// TIA Portal project "2020冬完善底层" (V15)

(* hardware
DEVICE "S7-1200 station_1"  S7-1200 Station
   slot 0: "Rack_0"  S7-1200 Rack  Rack  V1.0
   slot 1: "PLC_1"  CPU 1212C DC/DC/DC  6ES7 212-1AE40-0XB0  V4.2
   slot 3: "AQ 1x12BIT_1"  AQ1 signal board  6ES7 232-4HA30-0XB0  V1.0
DEVICE "S7-1200 station_2"  S7-1200 Station
   slot 0: "Rack_0"  S7-1200 Rack  Rack  V1.0
   slot 1: "PLC_2"  CPU 1212C DC/DC/DC  6ES7 212-1AE40-0XB0  V4.2
   slot 3: "AQ 1x12BIT_1"  AQ1 signal board  6ES7 232-4HA30-0XB0  V1.0
DEVICE "S7-1200 station_3"  S7-1200 Station
   slot 0: "Rack_0"  S7-1200 Rack  Rack  V1.0
   slot 1: "PLC_3"  CPU 1212C DC/DC/DC  6ES7 212-1AE40-0XB0  V4.2
   slot 3: "AQ 1x12BIT_1"  AQ1 signal board  6ES7 232-4HA30-0XB0  V1.0
DEVICE "S7-1200 station_4"  S7-1200 Station
   slot 0: "Rack_0"  S7-1200 Rack  Rack  V1.0
   slot 1: "PLC_4"  CPU 1212C DC/DC/DC  6ES7 212-1AE40-0XB0  V4.2
   slot 3: "AQ 1x12BIT_1"  AQ1 signal board  6ES7 232-4HA30-0XB0  V1.0
*)

// ===== PLC "PLC_1"  CPU 1212C DC/DC/DC =====

VAR_GLOBAL   // PLC tag table "默认变量表"
   "JogForward" AT %I200.0 : Bool;
   "JogBackward" AT %I200.1 : Bool;
   "driver" AT %I200.2 : Bool;
   "Anlonage input" AT %IW208 : Word;
   "R驱动编码器值" AT %ID1000 : DWord;
   "position" AT %IW202 : Word;
   "velecity" AT %ID204 : DWord;
   "R旋转编码器值" AT %ID1008 : DWord;
   "spin" AT %I200.3 : Bool;
   "轴_1_脉冲" AT %Q0.0 : Bool;
   "轴_1_方向" AT %Q0.1 : Bool;
   "AQ电压模拟量输出口" AT %QW80 : Word;
   "旋转编码器值保持" AT %MD0 : DWord;
   "一次写入" AT %M5.0 : Bool;
   "旋转速度转换real" AT %MD24 : Real;
   "原地转向临时速度" AT %MD100 : DWord;
   "原地转向-二号车轮转换" AT %MD104 : Real;
   "原地转向-四号车轮转换" AT %MD108 : Real;
   "原地转向-三号车轮转换" AT %MD112 : Real;
   "二号车轮方向判断继电器" AT %M118.0 : Bool;
   "三号车轮方向判断继电器" AT %M118.1 : Bool;
   "四号车轮方向判断继电器" AT %M118.2 : Bool;
END_VAR

DATA_BLOCK "数据块_1"   // DB1
{ S7_Optimized_Access := 'FALSE' }
VERSION : 0.1
   VAR
      一号车轮旋转开关 : Bool;
      一号车轮直行开关 : Bool;
      一号车轮目标旋转位置 : Word;
      一号车论旋转速度 : DWord;
      "一号车轮直行模拟量（已校准）" : Word;
      二号车轮旋转开关 : Bool;
      二号车轮直行开关 : Bool;
      二号车轮目标旋转位置 : Word;
      二号车轮旋转速度 : DWord;
      "二号车轮直行模拟量（已校准）" : Word;
      三号车轮旋转开关 : Bool;
      三号车轮直行开关 : Bool;
      三号车轮目标旋转位置 : Word;
      三号车轮旋转速度 : DWord;
      "三号车轮直行模拟量（已校准）" : Word;
      四号车轮旋转开关 : Bool;
      四号车轮直行开关 : Bool;
      四号车轮目标旋转位置 : Word;
      四号车轮旋转速度 : DWord;
      "四号车轮直行模拟量（已校准）" : Word;
      "转弯半径（未用）" : Int;
      运动模式 : Byte;
      一号车轮转角编码器读取 : DWord;
      一号车轮速度编码器读取 : DWord;
      二号车轮转角编码器读取 : DWord;
      二号车轮速度编码器读取 : DWord;
      三号车轮转角编码器读取 : DWord;
      三号车轮速度编码器读取 : DWord;
      四号车轮转角编码器读取 : DWord;
      四号车轮速度编码器读取 : DWord;
      一号车轮写入速度 : Word;
      二号车轮写入速度 : Word;
      三号车轮写入速度 : Word;
      四号车轮写入速度 : Word;
   END_VAR
BEGIN
END_DATA_BLOCK

DATA_BLOCK "轴_1"   // DB2, Motion_DB
{ S7_Optimized_Access := 'TRUE' }
AUTHOR : SIMATIC
FAMILY : BasicMC
NAME : TO_PosAx
VERSION : 6.0
// stored: InstanceOfName TO_PositioningAxis
"TO_PositioningAxis"
BEGIN
   // Axis.OnlinePtoModeCU = 16#0000_0002
   // Axis.DirectionOutputEnabledCU = TRUE
   // Axis.SelectedChannel2EnumCU = %Q0.1
   // Axis.SelectedChannel1EnumCU = %Q0.0
   // Pulse.MinDeltaDeltaFrequencyCU = 0.004
   // Pulse.MaxDeltaDeltaFrequencyCU = 1.0E+10
   // Pulse.MinDeltaFrequencyCU = 0.005
   // Pulse.MaxDeltaFrequencyCU = 9.5E+9
   // Pulse.MinFrequencyCU = 1.0
   // Pulse.MaxFrequencyCU = 100000.0
   // Pulse.OutputSourceCU = 16#0000_0000
   // Axis.SelectPTO = 0
END_DATA_BLOCK

FUNCTION "WRITE设备数据传递到各个设备" : Void   // FC1, SCL
{ S7_Optimized_Access := 'TRUE' }
VERSION : 0.1
BEGIN
   POKE_BLK(area_src := 16#84,
            dbNumber_src := 1,
            byteOffset_src := 10,
            area_dest := 16#82,
            dbNumber_dest := 0,
            byteOffset_dest := 200,
            count := 30);
   POKE_BLK(area_src := 16#84,
            dbNumber_src := 1,
            byteOffset_src := 2,
            area_dest := 16#81,
            dbNumber_dest := 0,
            byteOffset_dest := 202,
            count := 8);
   POKE_BLK(area_src:=16#81,
            dbNumber_src:=0,
            byteOffset_src:=300,
            area_dest:=16#84,
            dbNumber_dest:=1,
            byteOffset_dest:=52,
            count:=24);
END_FUNCTION

FUNCTION "模式选择" : Void   // FC2, LAD
{ S7_Optimized_Access := 'TRUE' }
VERSION : 0.1
BEGIN

REGION Network 1
   // 运动模式，01为四轮02为四轮异向03为前轮04为原地
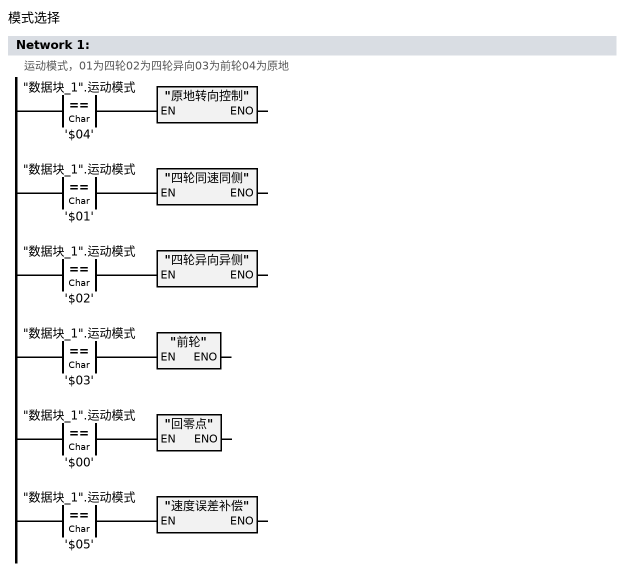
   RUNG wire#powerrail
      { S7_Templates := "SrcType := Char" } EQ_Contact(in1 := "数据块_1".运动模式, in2 := '$04')
      "原地转向控制"()
   END_RUNG
   RUNG wire#powerrail
      { S7_Templates := "SrcType := Char" } EQ_Contact(in1 := "数据块_1".运动模式, in2 := '$01')
      "四轮同速同侧"()
   END_RUNG
   RUNG wire#powerrail
      { S7_Templates := "SrcType := Char" } EQ_Contact(in1 := "数据块_1".运动模式, in2 := '$02')
      "四轮异向异侧"()
   END_RUNG
   RUNG wire#powerrail
      { S7_Templates := "SrcType := Char" } EQ_Contact(in1 := "数据块_1".运动模式, in2 := '$03')
      "前轮"()
   END_RUNG
   RUNG wire#powerrail
      { S7_Templates := "SrcType := Char" } EQ_Contact(in1 := "数据块_1".运动模式, in2 := '$00')
      "回零点"()
   END_RUNG
   RUNG wire#powerrail
      { S7_Templates := "SrcType := Char" } EQ_Contact(in1 := "数据块_1".运动模式, in2 := '$05')
      "速度误差补偿"()
   END_RUNG
   // the same network as SCL:
   IF "数据块_1".运动模式 = '$04' THEN "原地转向控制"(); END_IF;
   IF "数据块_1".运动模式 = '$01' THEN "四轮同速同侧"(); END_IF;
   IF "数据块_1".运动模式 = '$02' THEN "四轮异向异侧"(); END_IF;
   IF "数据块_1".运动模式 = '$03' THEN "前轮"(); END_IF;
   IF "数据块_1".运动模式 = '$00' THEN "回零点"(); END_IF;
   IF "数据块_1".运动模式 = '$05' THEN "速度误差补偿"(); END_IF;
END_REGION
END_FUNCTION

FUNCTION "原地转向控制" : Void   // FC3, LAD
{ S7_Optimized_Access := 'TRUE' }
VERSION : 0.1
BEGIN

REGION Network 1
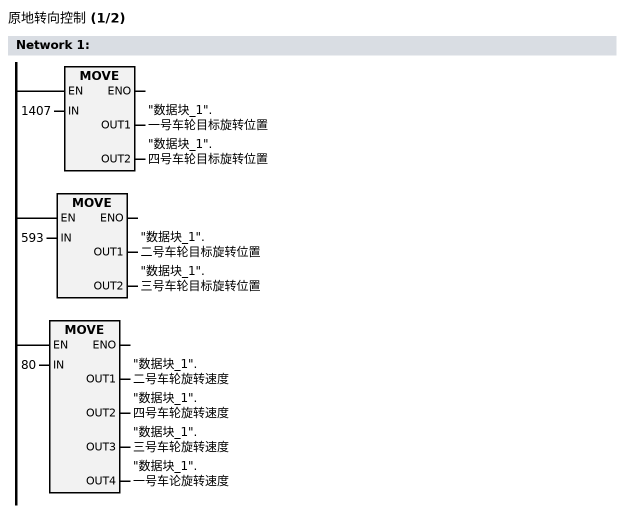
   RUNG wire#powerrail
      Move(in := 1407, out1 => "数据块_1".一号车轮目标旋转位置, out2 => "数据块_1".四号车轮目标旋转位置)
   END_RUNG
   RUNG wire#powerrail
      Move(in := 593, out1 => "数据块_1".二号车轮目标旋转位置, out2 => "数据块_1".三号车轮目标旋转位置)
   END_RUNG
   RUNG wire#powerrail
      Move(in := 80, out1 => "数据块_1".二号车轮旋转速度, out2 => "数据块_1".四号车轮旋转速度, out3 => "数据块_1".三号车轮旋转速度, out4 => "数据块_1".一号车论旋转速度)
   END_RUNG
   // the same network as SCL:
   "数据块_1".一号车轮目标旋转位置 := 1407;
   "数据块_1".四号车轮目标旋转位置 := 1407;
   "数据块_1".二号车轮目标旋转位置 := 593;
   "数据块_1".三号车轮目标旋转位置 := 593;
   "数据块_1".二号车轮旋转速度 := 80;
   "数据块_1".四号车轮旋转速度 := 80;
   "数据块_1".三号车轮旋转速度 := 80;
   "数据块_1".一号车论旋转速度 := 80;
END_REGION

REGION Network 2
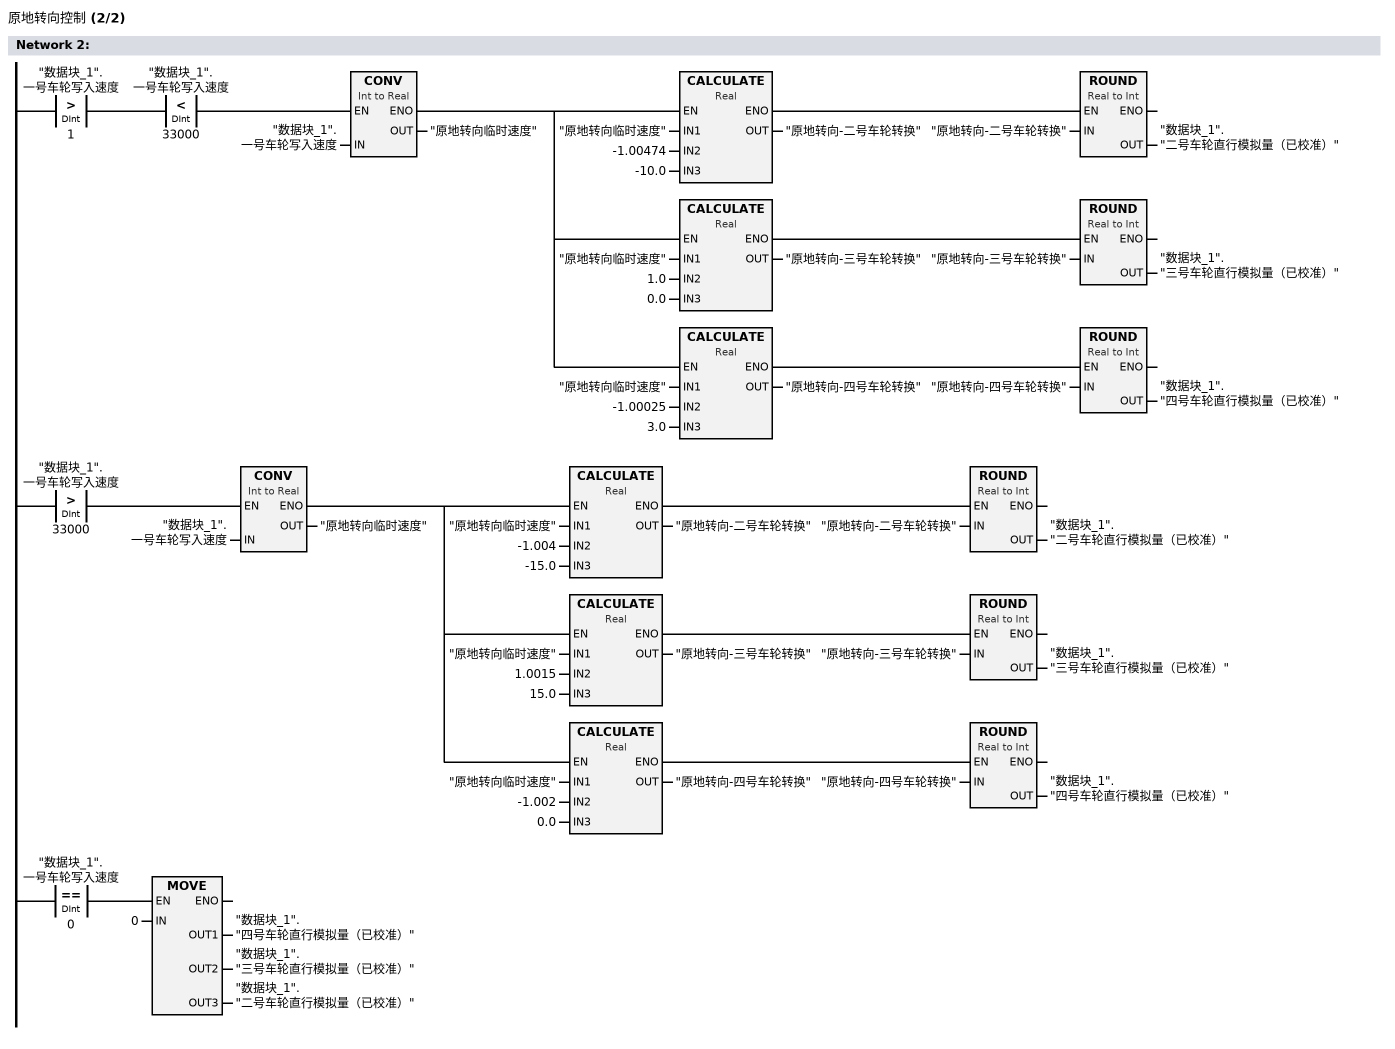
   RUNG wire#powerrail
      { S7_Templates := "SrcType := DInt" } GT_Contact(in1 := "数据块_1".一号车轮写入速度, in2 := 1)
      { S7_Templates := "SrcType := DInt" } LT_Contact(in1 := "数据块_1".一号车轮写入速度, in2 := 33000)
      { S7_Templates := "[SrcType := Int, DestType := Real]" } Convert(in := "数据块_1".一号车轮写入速度, out => "原地转向临时速度")
      wire#w1
      { S7_Templates := "SrcType := Real"; S7_Expression := "IN1*IN2+IN3" } Calculate(in1 := "原地转向临时速度", in2 := -1.00474, in3 := -10.0, out => "原地转向-二号车轮转换")
      { S7_Templates := "[SrcType := Real, DestType := Int]" } Round(in := "原地转向-二号车轮转换", out => "数据块_1"."二号车轮直行模拟量（已校准）")
   END_RUNG
   RUNG wire#w1
      { S7_Templates := "SrcType := Real"; S7_Expression := "IN1*IN2+IN3" } Calculate(in1 := "原地转向临时速度", in2 := 1.0, in3 := 0.0, out => "原地转向-三号车轮转换")
      { S7_Templates := "[SrcType := Real, DestType := Int]" } Round(in := "原地转向-三号车轮转换", out => "数据块_1"."三号车轮直行模拟量（已校准）")
   END_RUNG
   RUNG wire#w1
      { S7_Templates := "SrcType := Real"; S7_Expression := "IN1*IN2+IN3" } Calculate(in1 := "原地转向临时速度", in2 := -1.00025, in3 := 3.0, out => "原地转向-四号车轮转换")
      { S7_Templates := "[SrcType := Real, DestType := Int]" } Round(in := "原地转向-四号车轮转换", out => "数据块_1"."四号车轮直行模拟量（已校准）")
   END_RUNG
   RUNG wire#powerrail
      { S7_Templates := "SrcType := DInt" } GT_Contact(in1 := "数据块_1".一号车轮写入速度, in2 := 33000)
      { S7_Templates := "[SrcType := Int, DestType := Real]" } Convert(in := "数据块_1".一号车轮写入速度, out => "原地转向临时速度")
      wire#w2
      { S7_Templates := "SrcType := Real"; S7_Expression := "IN1*IN2+IN3" } Calculate(in1 := "原地转向临时速度", in2 := -1.004, in3 := -15.0, out => "原地转向-二号车轮转换")
      { S7_Templates := "[SrcType := Real, DestType := Int]" } Round(in := "原地转向-二号车轮转换", out => "数据块_1"."二号车轮直行模拟量（已校准）")
   END_RUNG
   RUNG wire#w2
      { S7_Templates := "SrcType := Real"; S7_Expression := "IN1*IN2+IN3" } Calculate(in1 := "原地转向临时速度", in2 := 1.0015, in3 := 15.0, out => "原地转向-三号车轮转换")
      { S7_Templates := "[SrcType := Real, DestType := Int]" } Round(in := "原地转向-三号车轮转换", out => "数据块_1"."三号车轮直行模拟量（已校准）")
   END_RUNG
   RUNG wire#w2
      { S7_Templates := "SrcType := Real"; S7_Expression := "IN1*IN2+IN3" } Calculate(in1 := "原地转向临时速度", in2 := -1.002, in3 := 0.0, out => "原地转向-四号车轮转换")
      { S7_Templates := "[SrcType := Real, DestType := Int]" } Round(in := "原地转向-四号车轮转换", out => "数据块_1"."四号车轮直行模拟量（已校准）")
   END_RUNG
   RUNG wire#powerrail
      { S7_Templates := "SrcType := DInt" } EQ_Contact(in1 := "数据块_1".一号车轮写入速度, in2 := 0)
      Move(in := 0, out1 => "数据块_1"."四号车轮直行模拟量（已校准）", out2 => "数据块_1"."三号车轮直行模拟量（已校准）", out3 => "数据块_1"."二号车轮直行模拟量（已校准）")
   END_RUNG
   // the same network as SCL:
   IF ("数据块_1".一号车轮写入速度 > 1) AND ("数据块_1".一号车轮写入速度 < 33000) THEN
       "原地转向临时速度" := INT_TO_REAL("数据块_1".一号车轮写入速度);
       "原地转向-二号车轮转换" := "原地转向临时速度"*(-1.00474)+(-10.0);
       "数据块_1"."二号车轮直行模拟量（已校准）" := ROUND("原地转向-二号车轮转换");
       "原地转向-三号车轮转换" := "原地转向临时速度"*1.0+0.0;
       "数据块_1"."三号车轮直行模拟量（已校准）" := ROUND("原地转向-三号车轮转换");
       "原地转向-四号车轮转换" := "原地转向临时速度"*(-1.00025)+3.0;
       "数据块_1"."四号车轮直行模拟量（已校准）" := ROUND("原地转向-四号车轮转换");
   END_IF;
   IF "数据块_1".一号车轮写入速度 > 33000 THEN
       "原地转向临时速度" := INT_TO_REAL("数据块_1".一号车轮写入速度);
       "原地转向-二号车轮转换" := "原地转向临时速度"*(-1.004)+(-15.0);
       "数据块_1"."二号车轮直行模拟量（已校准）" := ROUND("原地转向-二号车轮转换");
       "原地转向-三号车轮转换" := "原地转向临时速度"*1.0015+15.0;
       "数据块_1"."三号车轮直行模拟量（已校准）" := ROUND("原地转向-三号车轮转换");
       "原地转向-四号车轮转换" := "原地转向临时速度"*(-1.002)+0.0;
       "数据块_1"."四号车轮直行模拟量（已校准）" := ROUND("原地转向-四号车轮转换");
   END_IF;
   IF "数据块_1".一号车轮写入速度 = 0 THEN
       "数据块_1"."四号车轮直行模拟量（已校准）" := 0;
       "数据块_1"."三号车轮直行模拟量（已校准）" := 0;
       "数据块_1"."二号车轮直行模拟量（已校准）" := 0;
   END_IF;
END_REGION
END_FUNCTION

FUNCTION "四轮同速同侧" : Void   // FC5, LAD
{ S7_Optimized_Access := 'TRUE' }
VERSION : 0.1
BEGIN

REGION Network 1
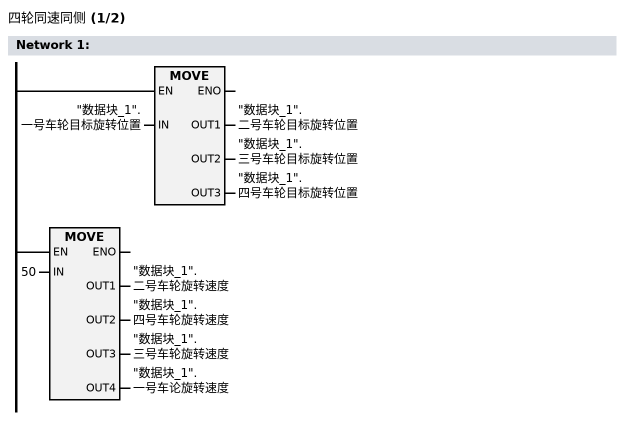
   RUNG wire#powerrail
      Move(in := "数据块_1".一号车轮目标旋转位置, out1 => "数据块_1".二号车轮目标旋转位置, out2 => "数据块_1".三号车轮目标旋转位置, out3 => "数据块_1".四号车轮目标旋转位置)
   END_RUNG
   RUNG wire#powerrail
      Move(in := 50, out1 => "数据块_1".二号车轮旋转速度, out2 => "数据块_1".四号车轮旋转速度, out3 => "数据块_1".三号车轮旋转速度, out4 => "数据块_1".一号车论旋转速度)
   END_RUNG
   // the same network as SCL:
   "数据块_1".二号车轮目标旋转位置 := "数据块_1".一号车轮目标旋转位置;
   "数据块_1".三号车轮目标旋转位置 := "数据块_1".一号车轮目标旋转位置;
   "数据块_1".四号车轮目标旋转位置 := "数据块_1".一号车轮目标旋转位置;
   "数据块_1".二号车轮旋转速度 := 50;
   "数据块_1".四号车轮旋转速度 := 50;
   "数据块_1".三号车轮旋转速度 := 50;
   "数据块_1".一号车论旋转速度 := 50;
END_REGION

REGION Network 2
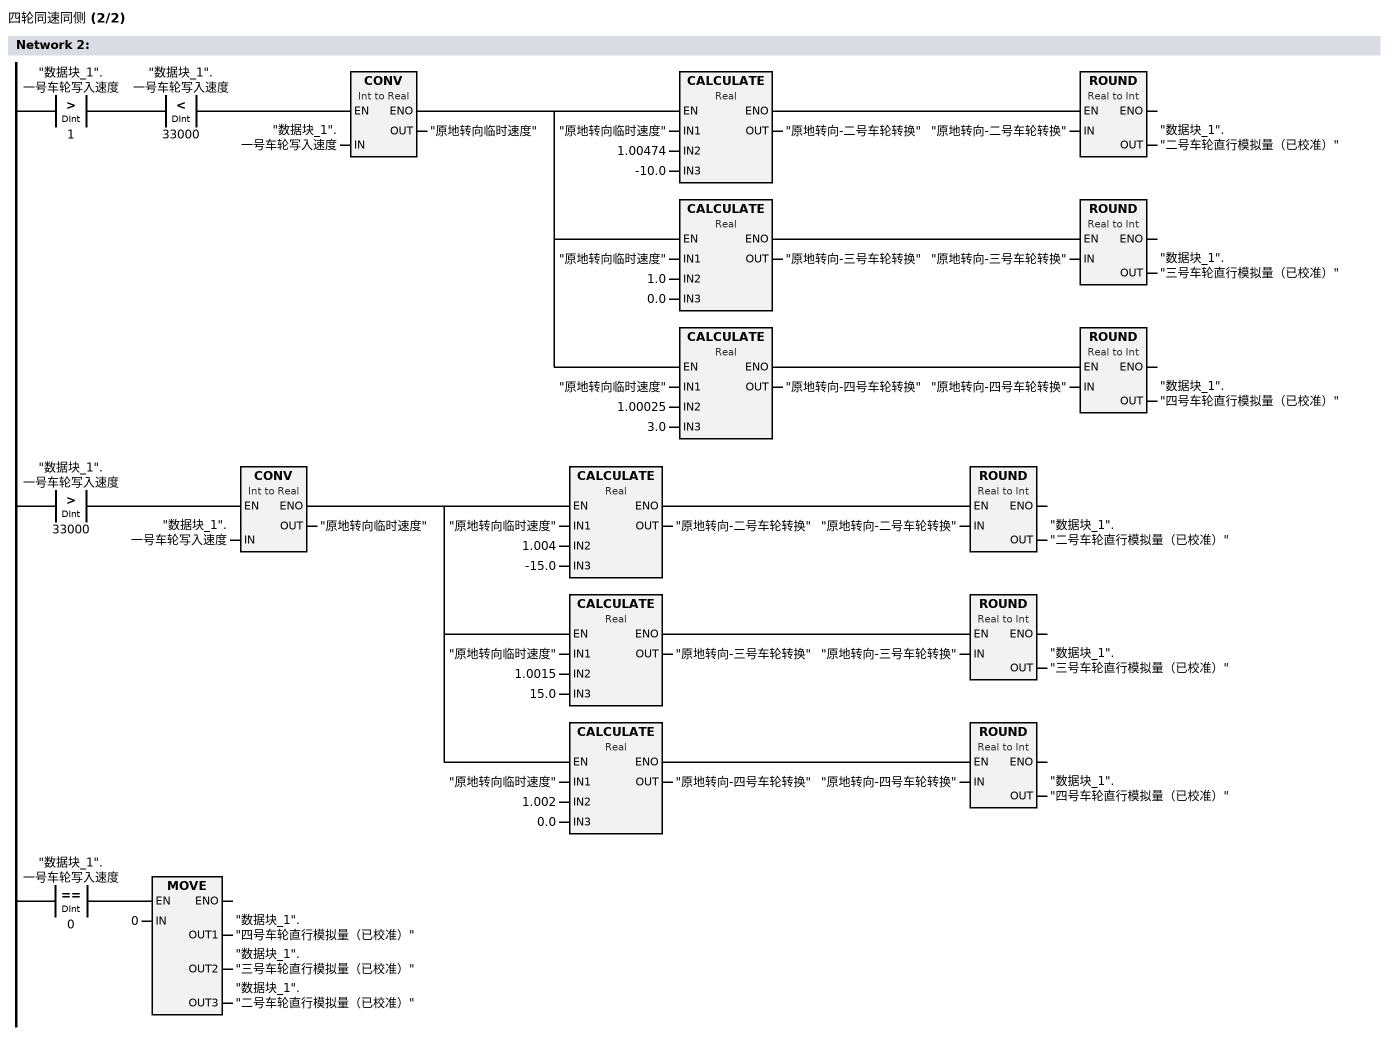
   RUNG wire#powerrail
      { S7_Templates := "SrcType := DInt" } GT_Contact(in1 := "数据块_1".一号车轮写入速度, in2 := 1)
      { S7_Templates := "SrcType := DInt" } LT_Contact(in1 := "数据块_1".一号车轮写入速度, in2 := 33000)
      { S7_Templates := "[SrcType := Int, DestType := Real]" } Convert(in := "数据块_1".一号车轮写入速度, out => "原地转向临时速度")
      wire#w1
      { S7_Templates := "SrcType := Real"; S7_Expression := "IN1*IN2+IN3" } Calculate(in1 := "原地转向临时速度", in2 := 1.00474, in3 := -10.0, out => "原地转向-二号车轮转换")
      { S7_Templates := "[SrcType := Real, DestType := Int]" } Round(in := "原地转向-二号车轮转换", out => "数据块_1"."二号车轮直行模拟量（已校准）")
   END_RUNG
   RUNG wire#w1
      { S7_Templates := "SrcType := Real"; S7_Expression := "IN1*IN2+IN3" } Calculate(in1 := "原地转向临时速度", in2 := 1.0, in3 := 0.0, out => "原地转向-三号车轮转换")
      { S7_Templates := "[SrcType := Real, DestType := Int]" } Round(in := "原地转向-三号车轮转换", out => "数据块_1"."三号车轮直行模拟量（已校准）")
   END_RUNG
   RUNG wire#w1
      { S7_Templates := "SrcType := Real"; S7_Expression := "IN1*IN2+IN3" } Calculate(in1 := "原地转向临时速度", in2 := 1.00025, in3 := 3.0, out => "原地转向-四号车轮转换")
      { S7_Templates := "[SrcType := Real, DestType := Int]" } Round(in := "原地转向-四号车轮转换", out => "数据块_1"."四号车轮直行模拟量（已校准）")
   END_RUNG
   RUNG wire#powerrail
      { S7_Templates := "SrcType := DInt" } GT_Contact(in1 := "数据块_1".一号车轮写入速度, in2 := 33000)
      { S7_Templates := "[SrcType := Int, DestType := Real]" } Convert(in := "数据块_1".一号车轮写入速度, out => "原地转向临时速度")
      wire#w2
      { S7_Templates := "SrcType := Real"; S7_Expression := "IN1*IN2+IN3" } Calculate(in1 := "原地转向临时速度", in2 := 1.004, in3 := -15.0, out => "原地转向-二号车轮转换")
      { S7_Templates := "[SrcType := Real, DestType := Int]" } Round(in := "原地转向-二号车轮转换", out => "数据块_1"."二号车轮直行模拟量（已校准）")
   END_RUNG
   RUNG wire#w2
      { S7_Templates := "SrcType := Real"; S7_Expression := "IN1*IN2+IN3" } Calculate(in1 := "原地转向临时速度", in2 := 1.0015, in3 := 15.0, out => "原地转向-三号车轮转换")
      { S7_Templates := "[SrcType := Real, DestType := Int]" } Round(in := "原地转向-三号车轮转换", out => "数据块_1"."三号车轮直行模拟量（已校准）")
   END_RUNG
   RUNG wire#w2
      { S7_Templates := "SrcType := Real"; S7_Expression := "IN1*IN2+IN3" } Calculate(in1 := "原地转向临时速度", in2 := 1.002, in3 := 0.0, out => "原地转向-四号车轮转换")
      { S7_Templates := "[SrcType := Real, DestType := Int]" } Round(in := "原地转向-四号车轮转换", out => "数据块_1"."四号车轮直行模拟量（已校准）")
   END_RUNG
   RUNG wire#powerrail
      { S7_Templates := "SrcType := DInt" } EQ_Contact(in1 := "数据块_1".一号车轮写入速度, in2 := 0)
      Move(in := 0, out1 => "数据块_1"."四号车轮直行模拟量（已校准）", out2 => "数据块_1"."三号车轮直行模拟量（已校准）", out3 => "数据块_1"."二号车轮直行模拟量（已校准）")
   END_RUNG
   // the same network as SCL:
   IF ("数据块_1".一号车轮写入速度 > 1) AND ("数据块_1".一号车轮写入速度 < 33000) THEN
       "原地转向临时速度" := INT_TO_REAL("数据块_1".一号车轮写入速度);
       "原地转向-二号车轮转换" := "原地转向临时速度"*1.00474+(-10.0);
       "数据块_1"."二号车轮直行模拟量（已校准）" := ROUND("原地转向-二号车轮转换");
       "原地转向-三号车轮转换" := "原地转向临时速度"*1.0+0.0;
       "数据块_1"."三号车轮直行模拟量（已校准）" := ROUND("原地转向-三号车轮转换");
       "原地转向-四号车轮转换" := "原地转向临时速度"*1.00025+3.0;
       "数据块_1"."四号车轮直行模拟量（已校准）" := ROUND("原地转向-四号车轮转换");
   END_IF;
   IF "数据块_1".一号车轮写入速度 > 33000 THEN
       "原地转向临时速度" := INT_TO_REAL("数据块_1".一号车轮写入速度);
       "原地转向-二号车轮转换" := "原地转向临时速度"*1.004+(-15.0);
       "数据块_1"."二号车轮直行模拟量（已校准）" := ROUND("原地转向-二号车轮转换");
       "原地转向-三号车轮转换" := "原地转向临时速度"*1.0015+15.0;
       "数据块_1"."三号车轮直行模拟量（已校准）" := ROUND("原地转向-三号车轮转换");
       "原地转向-四号车轮转换" := "原地转向临时速度"*1.002+0.0;
       "数据块_1"."四号车轮直行模拟量（已校准）" := ROUND("原地转向-四号车轮转换");
   END_IF;
   IF "数据块_1".一号车轮写入速度 = 0 THEN
       "数据块_1"."四号车轮直行模拟量（已校准）" := 0;
       "数据块_1"."三号车轮直行模拟量（已校准）" := 0;
       "数据块_1"."二号车轮直行模拟量（已校准）" := 0;
   END_IF;
END_REGION
END_FUNCTION

FUNCTION "四轮异向异侧" : Void   // FC6, LAD
{ S7_Optimized_Access := 'TRUE' }
VERSION : 0.1
BEGIN

REGION Network 1
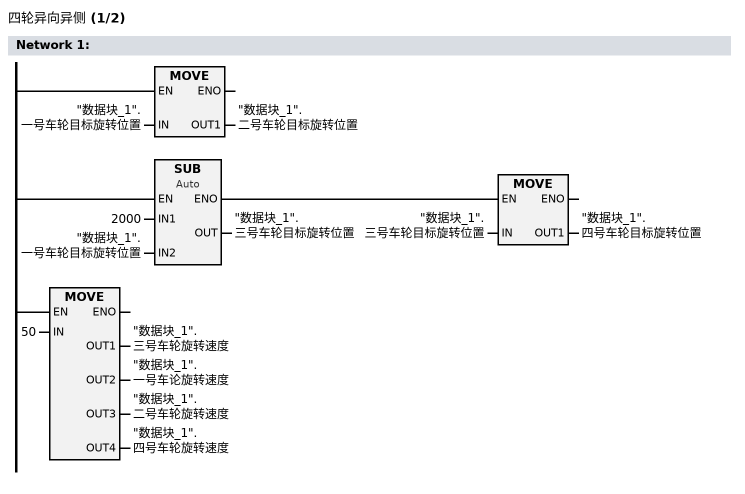
   RUNG wire#powerrail
      Move(in := "数据块_1".一号车轮目标旋转位置, out1 => "数据块_1".二号车轮目标旋转位置)
   END_RUNG
   RUNG wire#powerrail
      Sub(in1 := 2000, in2 := "数据块_1".一号车轮目标旋转位置, out => "数据块_1".三号车轮目标旋转位置)
      Move(in := "数据块_1".三号车轮目标旋转位置, out1 => "数据块_1".四号车轮目标旋转位置)
   END_RUNG
   RUNG wire#powerrail
      Move(in := 50, out1 => "数据块_1".三号车轮旋转速度, out2 => "数据块_1".一号车论旋转速度, out3 => "数据块_1".二号车轮旋转速度, out4 => "数据块_1".四号车轮旋转速度)
   END_RUNG
   // the same network as SCL:
   "数据块_1".二号车轮目标旋转位置 := "数据块_1".一号车轮目标旋转位置;
   "数据块_1".三号车轮目标旋转位置 := 2000 - "数据块_1".一号车轮目标旋转位置;
   "数据块_1".四号车轮目标旋转位置 := "数据块_1".三号车轮目标旋转位置;
   "数据块_1".三号车轮旋转速度 := 50;
   "数据块_1".一号车论旋转速度 := 50;
   "数据块_1".二号车轮旋转速度 := 50;
   "数据块_1".四号车轮旋转速度 := 50;
END_REGION

REGION Network 2
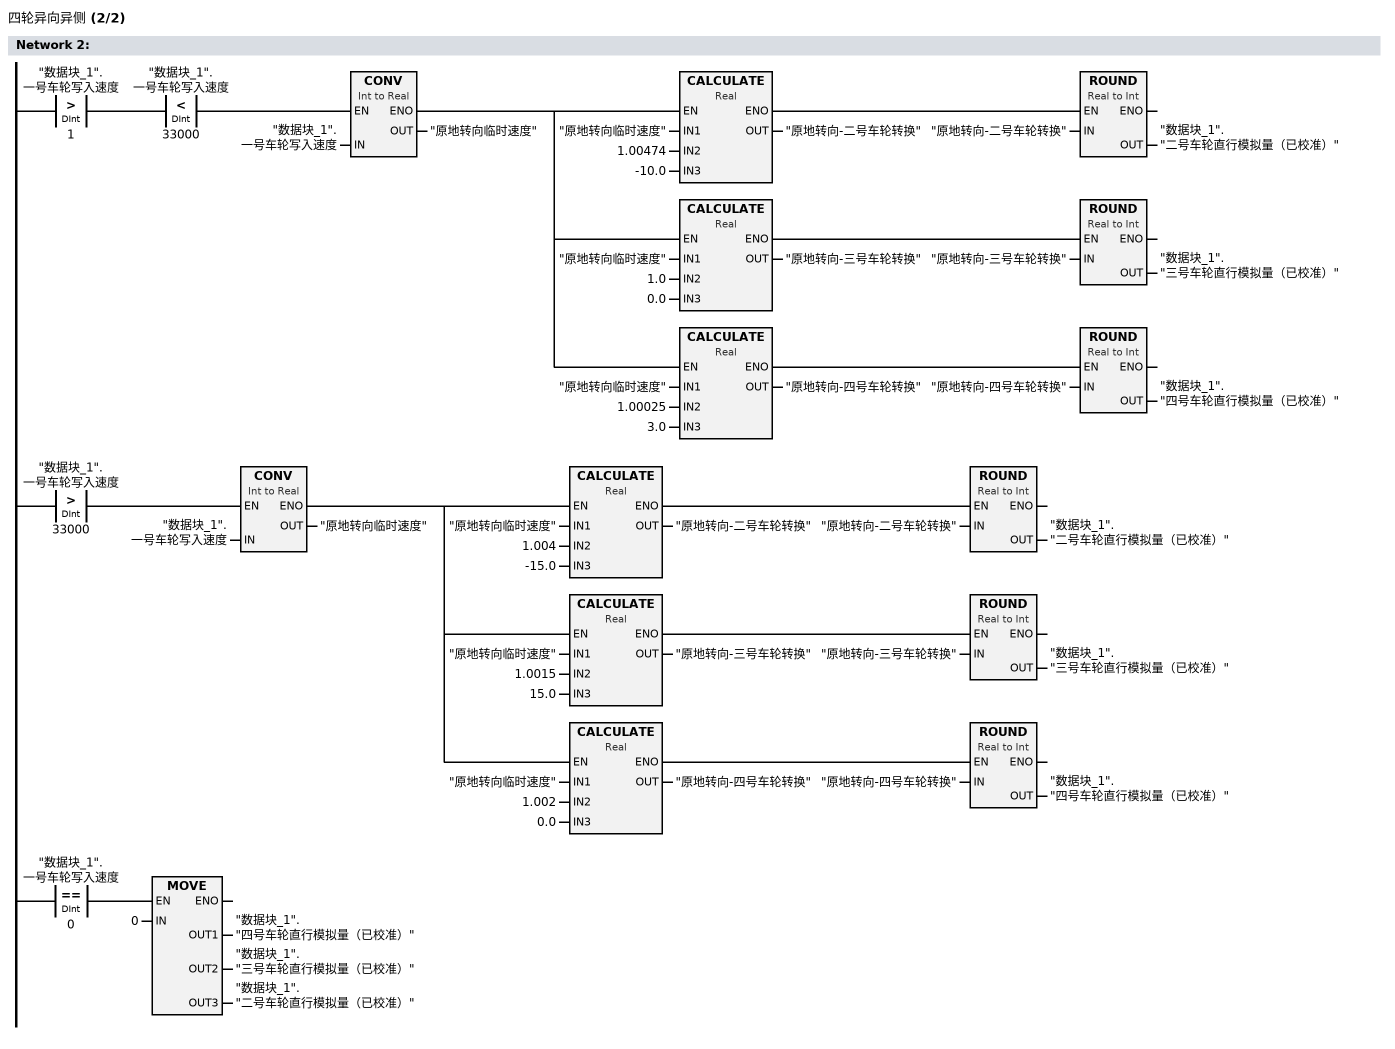
   RUNG wire#powerrail
      { S7_Templates := "SrcType := DInt" } GT_Contact(in1 := "数据块_1".一号车轮写入速度, in2 := 1)
      { S7_Templates := "SrcType := DInt" } LT_Contact(in1 := "数据块_1".一号车轮写入速度, in2 := 33000)
      { S7_Templates := "[SrcType := Int, DestType := Real]" } Convert(in := "数据块_1".一号车轮写入速度, out => "原地转向临时速度")
      wire#w1
      { S7_Templates := "SrcType := Real"; S7_Expression := "IN1*IN2+IN3" } Calculate(in1 := "原地转向临时速度", in2 := 1.00474, in3 := -10.0, out => "原地转向-二号车轮转换")
      { S7_Templates := "[SrcType := Real, DestType := Int]" } Round(in := "原地转向-二号车轮转换", out => "数据块_1"."二号车轮直行模拟量（已校准）")
   END_RUNG
   RUNG wire#w1
      { S7_Templates := "SrcType := Real"; S7_Expression := "IN1*IN2+IN3" } Calculate(in1 := "原地转向临时速度", in2 := 1.0, in3 := 0.0, out => "原地转向-三号车轮转换")
      { S7_Templates := "[SrcType := Real, DestType := Int]" } Round(in := "原地转向-三号车轮转换", out => "数据块_1"."三号车轮直行模拟量（已校准）")
   END_RUNG
   RUNG wire#w1
      { S7_Templates := "SrcType := Real"; S7_Expression := "IN1*IN2+IN3" } Calculate(in1 := "原地转向临时速度", in2 := 1.00025, in3 := 3.0, out => "原地转向-四号车轮转换")
      { S7_Templates := "[SrcType := Real, DestType := Int]" } Round(in := "原地转向-四号车轮转换", out => "数据块_1"."四号车轮直行模拟量（已校准）")
   END_RUNG
   RUNG wire#powerrail
      { S7_Templates := "SrcType := DInt" } GT_Contact(in1 := "数据块_1".一号车轮写入速度, in2 := 33000)
      { S7_Templates := "[SrcType := Int, DestType := Real]" } Convert(in := "数据块_1".一号车轮写入速度, out => "原地转向临时速度")
      wire#w2
      { S7_Templates := "SrcType := Real"; S7_Expression := "IN1*IN2+IN3" } Calculate(in1 := "原地转向临时速度", in2 := 1.004, in3 := -15.0, out => "原地转向-二号车轮转换")
      { S7_Templates := "[SrcType := Real, DestType := Int]" } Round(in := "原地转向-二号车轮转换", out => "数据块_1"."二号车轮直行模拟量（已校准）")
   END_RUNG
   RUNG wire#w2
      { S7_Templates := "SrcType := Real"; S7_Expression := "IN1*IN2+IN3" } Calculate(in1 := "原地转向临时速度", in2 := 1.0015, in3 := 15.0, out => "原地转向-三号车轮转换")
      { S7_Templates := "[SrcType := Real, DestType := Int]" } Round(in := "原地转向-三号车轮转换", out => "数据块_1"."三号车轮直行模拟量（已校准）")
   END_RUNG
   RUNG wire#w2
      { S7_Templates := "SrcType := Real"; S7_Expression := "IN1*IN2+IN3" } Calculate(in1 := "原地转向临时速度", in2 := 1.002, in3 := 0.0, out => "原地转向-四号车轮转换")
      { S7_Templates := "[SrcType := Real, DestType := Int]" } Round(in := "原地转向-四号车轮转换", out => "数据块_1"."四号车轮直行模拟量（已校准）")
   END_RUNG
   RUNG wire#powerrail
      { S7_Templates := "SrcType := DInt" } EQ_Contact(in1 := "数据块_1".一号车轮写入速度, in2 := 0)
      Move(in := 0, out1 => "数据块_1"."四号车轮直行模拟量（已校准）", out2 => "数据块_1"."三号车轮直行模拟量（已校准）", out3 => "数据块_1"."二号车轮直行模拟量（已校准）")
   END_RUNG
   // the same network as SCL:
   IF ("数据块_1".一号车轮写入速度 > 1) AND ("数据块_1".一号车轮写入速度 < 33000) THEN
       "原地转向临时速度" := INT_TO_REAL("数据块_1".一号车轮写入速度);
       "原地转向-二号车轮转换" := "原地转向临时速度"*1.00474+(-10.0);
       "数据块_1"."二号车轮直行模拟量（已校准）" := ROUND("原地转向-二号车轮转换");
       "原地转向-三号车轮转换" := "原地转向临时速度"*1.0+0.0;
       "数据块_1"."三号车轮直行模拟量（已校准）" := ROUND("原地转向-三号车轮转换");
       "原地转向-四号车轮转换" := "原地转向临时速度"*1.00025+3.0;
       "数据块_1"."四号车轮直行模拟量（已校准）" := ROUND("原地转向-四号车轮转换");
   END_IF;
   IF "数据块_1".一号车轮写入速度 > 33000 THEN
       "原地转向临时速度" := INT_TO_REAL("数据块_1".一号车轮写入速度);
       "原地转向-二号车轮转换" := "原地转向临时速度"*1.004+(-15.0);
       "数据块_1"."二号车轮直行模拟量（已校准）" := ROUND("原地转向-二号车轮转换");
       "原地转向-三号车轮转换" := "原地转向临时速度"*1.0015+15.0;
       "数据块_1"."三号车轮直行模拟量（已校准）" := ROUND("原地转向-三号车轮转换");
       "原地转向-四号车轮转换" := "原地转向临时速度"*1.002+0.0;
       "数据块_1"."四号车轮直行模拟量（已校准）" := ROUND("原地转向-四号车轮转换");
   END_IF;
   IF "数据块_1".一号车轮写入速度 = 0 THEN
       "数据块_1"."四号车轮直行模拟量（已校准）" := 0;
       "数据块_1"."三号车轮直行模拟量（已校准）" := 0;
       "数据块_1"."二号车轮直行模拟量（已校准）" := 0;
   END_IF;
END_REGION
END_FUNCTION

FUNCTION "前轮" : Void   // FC7, LAD
{ S7_Optimized_Access := 'TRUE' }
VERSION : 0.1
BEGIN

REGION Network 1
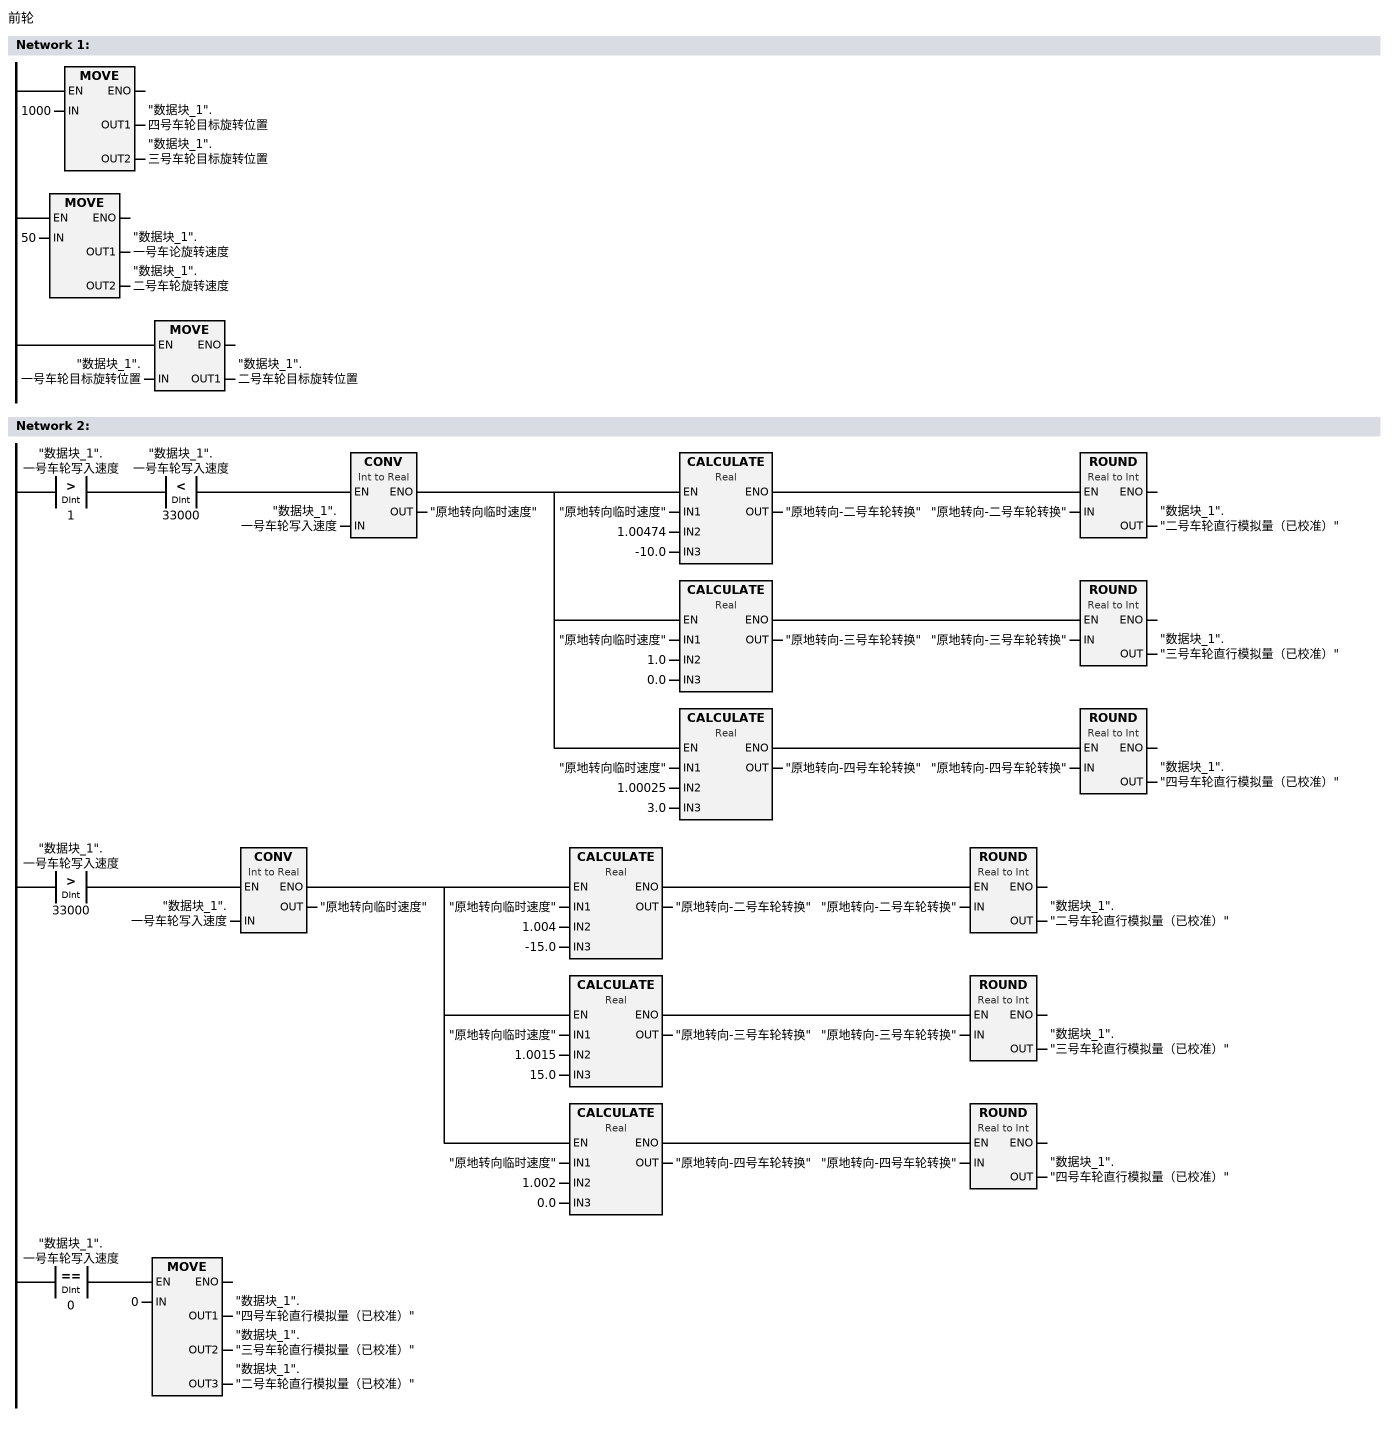
   RUNG wire#powerrail
      Move(in := 1000, out1 => "数据块_1".四号车轮目标旋转位置, out2 => "数据块_1".三号车轮目标旋转位置)
   END_RUNG
   RUNG wire#powerrail
      Move(in := 50, out1 => "数据块_1".一号车论旋转速度, out2 => "数据块_1".二号车轮旋转速度)
   END_RUNG
   RUNG wire#powerrail
      Move(in := "数据块_1".一号车轮目标旋转位置, out1 => "数据块_1".二号车轮目标旋转位置)
   END_RUNG
   // the same network as SCL:
   "数据块_1".四号车轮目标旋转位置 := 1000;
   "数据块_1".三号车轮目标旋转位置 := 1000;
   "数据块_1".一号车论旋转速度 := 50;
   "数据块_1".二号车轮旋转速度 := 50;
   "数据块_1".二号车轮目标旋转位置 := "数据块_1".一号车轮目标旋转位置;
END_REGION

REGION Network 2
   RUNG wire#powerrail
      { S7_Templates := "SrcType := DInt" } GT_Contact(in1 := "数据块_1".一号车轮写入速度, in2 := 1)
      { S7_Templates := "SrcType := DInt" } LT_Contact(in1 := "数据块_1".一号车轮写入速度, in2 := 33000)
      { S7_Templates := "[SrcType := Int, DestType := Real]" } Convert(in := "数据块_1".一号车轮写入速度, out => "原地转向临时速度")
      wire#w1
      { S7_Templates := "SrcType := Real"; S7_Expression := "IN1*IN2+IN3" } Calculate(in1 := "原地转向临时速度", in2 := 1.00474, in3 := -10.0, out => "原地转向-二号车轮转换")
      { S7_Templates := "[SrcType := Real, DestType := Int]" } Round(in := "原地转向-二号车轮转换", out => "数据块_1"."二号车轮直行模拟量（已校准）")
   END_RUNG
   RUNG wire#w1
      { S7_Templates := "SrcType := Real"; S7_Expression := "IN1*IN2+IN3" } Calculate(in1 := "原地转向临时速度", in2 := 1.0, in3 := 0.0, out => "原地转向-三号车轮转换")
      { S7_Templates := "[SrcType := Real, DestType := Int]" } Round(in := "原地转向-三号车轮转换", out => "数据块_1"."三号车轮直行模拟量（已校准）")
   END_RUNG
   RUNG wire#w1
      { S7_Templates := "SrcType := Real"; S7_Expression := "IN1*IN2+IN3" } Calculate(in1 := "原地转向临时速度", in2 := 1.00025, in3 := 3.0, out => "原地转向-四号车轮转换")
      { S7_Templates := "[SrcType := Real, DestType := Int]" } Round(in := "原地转向-四号车轮转换", out => "数据块_1"."四号车轮直行模拟量（已校准）")
   END_RUNG
   RUNG wire#powerrail
      { S7_Templates := "SrcType := DInt" } GT_Contact(in1 := "数据块_1".一号车轮写入速度, in2 := 33000)
      { S7_Templates := "[SrcType := Int, DestType := Real]" } Convert(in := "数据块_1".一号车轮写入速度, out => "原地转向临时速度")
      wire#w2
      { S7_Templates := "SrcType := Real"; S7_Expression := "IN1*IN2+IN3" } Calculate(in1 := "原地转向临时速度", in2 := 1.004, in3 := -15.0, out => "原地转向-二号车轮转换")
      { S7_Templates := "[SrcType := Real, DestType := Int]" } Round(in := "原地转向-二号车轮转换", out => "数据块_1"."二号车轮直行模拟量（已校准）")
   END_RUNG
   RUNG wire#w2
      { S7_Templates := "SrcType := Real"; S7_Expression := "IN1*IN2+IN3" } Calculate(in1 := "原地转向临时速度", in2 := 1.0015, in3 := 15.0, out => "原地转向-三号车轮转换")
      { S7_Templates := "[SrcType := Real, DestType := Int]" } Round(in := "原地转向-三号车轮转换", out => "数据块_1"."三号车轮直行模拟量（已校准）")
   END_RUNG
   RUNG wire#w2
      { S7_Templates := "SrcType := Real"; S7_Expression := "IN1*IN2+IN3" } Calculate(in1 := "原地转向临时速度", in2 := 1.002, in3 := 0.0, out => "原地转向-四号车轮转换")
      { S7_Templates := "[SrcType := Real, DestType := Int]" } Round(in := "原地转向-四号车轮转换", out => "数据块_1"."四号车轮直行模拟量（已校准）")
   END_RUNG
   RUNG wire#powerrail
      { S7_Templates := "SrcType := DInt" } EQ_Contact(in1 := "数据块_1".一号车轮写入速度, in2 := 0)
      Move(in := 0, out1 => "数据块_1"."四号车轮直行模拟量（已校准）", out2 => "数据块_1"."三号车轮直行模拟量（已校准）", out3 => "数据块_1"."二号车轮直行模拟量（已校准）")
   END_RUNG
   // the same network as SCL:
   IF ("数据块_1".一号车轮写入速度 > 1) AND ("数据块_1".一号车轮写入速度 < 33000) THEN
       "原地转向临时速度" := INT_TO_REAL("数据块_1".一号车轮写入速度);
       "原地转向-二号车轮转换" := "原地转向临时速度"*1.00474+(-10.0);
       "数据块_1"."二号车轮直行模拟量（已校准）" := ROUND("原地转向-二号车轮转换");
       "原地转向-三号车轮转换" := "原地转向临时速度"*1.0+0.0;
       "数据块_1"."三号车轮直行模拟量（已校准）" := ROUND("原地转向-三号车轮转换");
       "原地转向-四号车轮转换" := "原地转向临时速度"*1.00025+3.0;
       "数据块_1"."四号车轮直行模拟量（已校准）" := ROUND("原地转向-四号车轮转换");
   END_IF;
   IF "数据块_1".一号车轮写入速度 > 33000 THEN
       "原地转向临时速度" := INT_TO_REAL("数据块_1".一号车轮写入速度);
       "原地转向-二号车轮转换" := "原地转向临时速度"*1.004+(-15.0);
       "数据块_1"."二号车轮直行模拟量（已校准）" := ROUND("原地转向-二号车轮转换");
       "原地转向-三号车轮转换" := "原地转向临时速度"*1.0015+15.0;
       "数据块_1"."三号车轮直行模拟量（已校准）" := ROUND("原地转向-三号车轮转换");
       "原地转向-四号车轮转换" := "原地转向临时速度"*1.002+0.0;
       "数据块_1"."四号车轮直行模拟量（已校准）" := ROUND("原地转向-四号车轮转换");
   END_IF;
   IF "数据块_1".一号车轮写入速度 = 0 THEN
       "数据块_1"."四号车轮直行模拟量（已校准）" := 0;
       "数据块_1"."三号车轮直行模拟量（已校准）" := 0;
       "数据块_1"."二号车轮直行模拟量（已校准）" := 0;
   END_IF;
END_REGION
END_FUNCTION

FUNCTION "速度误差补偿" : Void   // FC8, LAD
{ S7_Optimized_Access := 'TRUE' }
VERSION : 0.1
BEGIN

REGION Network 1
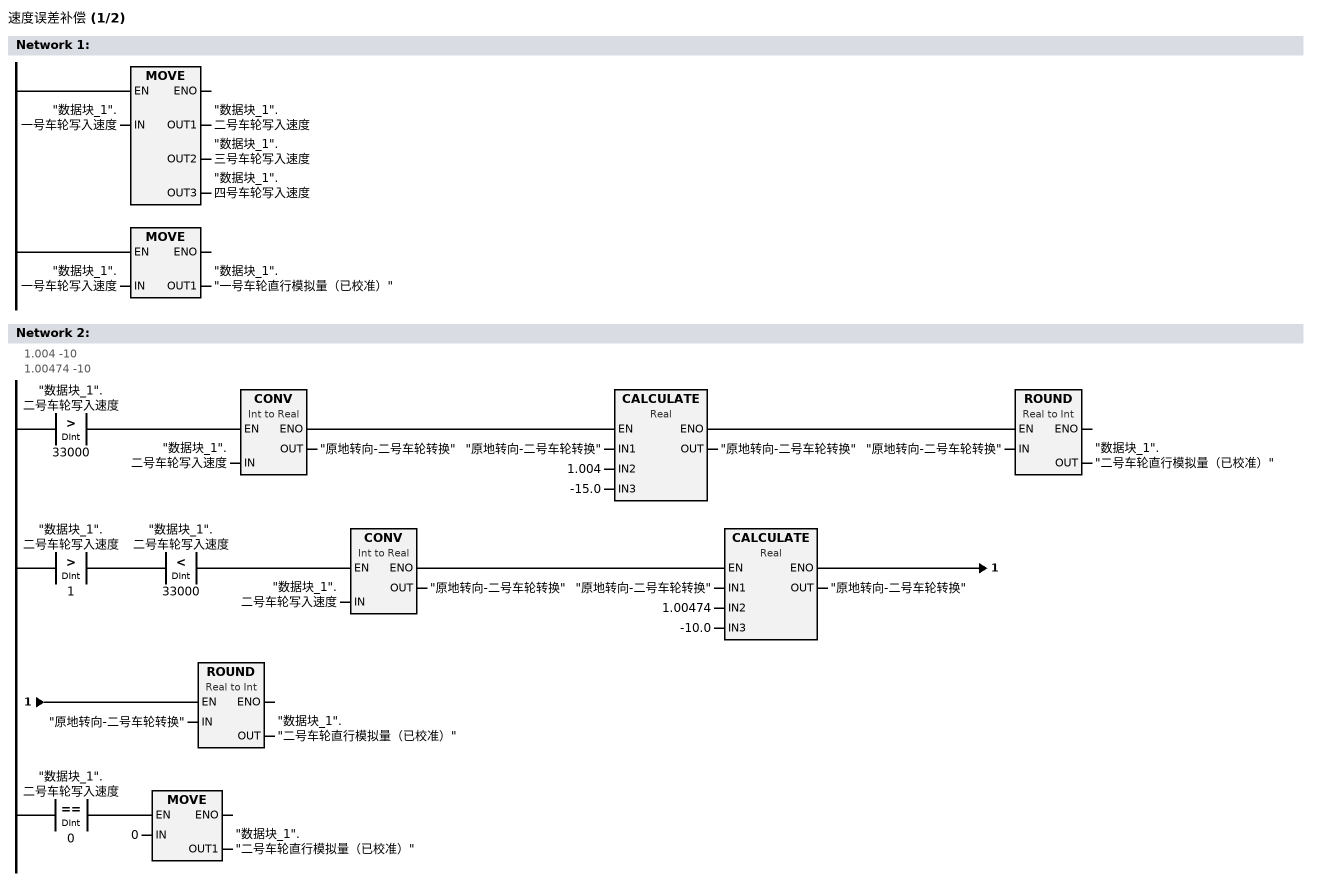
   RUNG wire#powerrail
      Move(in := "数据块_1".一号车轮写入速度, out1 => "数据块_1".二号车轮写入速度, out2 => "数据块_1".三号车轮写入速度, out3 => "数据块_1".四号车轮写入速度)
   END_RUNG
   RUNG wire#powerrail
      Move(in := "数据块_1".一号车轮写入速度, out1 => "数据块_1"."一号车轮直行模拟量（已校准）")
   END_RUNG
   // the same network as SCL:
   "数据块_1".二号车轮写入速度 := "数据块_1".一号车轮写入速度;
   "数据块_1".三号车轮写入速度 := "数据块_1".一号车轮写入速度;
   "数据块_1".四号车轮写入速度 := "数据块_1".一号车轮写入速度;
   "数据块_1"."一号车轮直行模拟量（已校准）" := "数据块_1".一号车轮写入速度;
END_REGION

REGION Network 2
   // 1.004 -10
   // 1.00474 -10
   RUNG wire#powerrail
      { S7_Templates := "SrcType := DInt" } GT_Contact(in1 := "数据块_1".二号车轮写入速度, in2 := 33000)
      { S7_Templates := "[SrcType := Int, DestType := Real]" } Convert(in := "数据块_1".二号车轮写入速度, out => "原地转向-二号车轮转换")
      { S7_Templates := "SrcType := Real"; S7_Expression := "IN1*IN2+IN3" } Calculate(in1 := "原地转向-二号车轮转换", in2 := 1.004, in3 := -15.0, out => "原地转向-二号车轮转换")
      { S7_Templates := "[SrcType := Real, DestType := Int]" } Round(in := "原地转向-二号车轮转换", out => "数据块_1"."二号车轮直行模拟量（已校准）")
   END_RUNG
   RUNG wire#powerrail
      { S7_Templates := "SrcType := DInt" } GT_Contact(in1 := "数据块_1".二号车轮写入速度, in2 := 1)
      { S7_Templates := "SrcType := DInt" } LT_Contact(in1 := "数据块_1".二号车轮写入速度, in2 := 33000)
      { S7_Templates := "[SrcType := Int, DestType := Real]" } Convert(in := "数据块_1".二号车轮写入速度, out => "原地转向-二号车轮转换")
      { S7_Templates := "SrcType := Real"; S7_Expression := "IN1*IN2+IN3" } Calculate(in1 := "原地转向-二号车轮转换", in2 := 1.00474, in3 := -10.0, out => "原地转向-二号车轮转换")
      { S7_Templates := "[SrcType := Real, DestType := Int]" } Round(in := "原地转向-二号车轮转换", out => "数据块_1"."二号车轮直行模拟量（已校准）")
   END_RUNG
   RUNG wire#powerrail
      { S7_Templates := "SrcType := DInt" } EQ_Contact(in1 := "数据块_1".二号车轮写入速度, in2 := 0)
      Move(in := 0, out1 => "数据块_1"."二号车轮直行模拟量（已校准）")
   END_RUNG
   // the same network as SCL:
   IF "数据块_1".二号车轮写入速度 > 33000 THEN
       "原地转向-二号车轮转换" := INT_TO_REAL("数据块_1".二号车轮写入速度);
       "原地转向-二号车轮转换" := "原地转向-二号车轮转换"*1.004+(-15.0);
       "数据块_1"."二号车轮直行模拟量（已校准）" := ROUND("原地转向-二号车轮转换");
   END_IF;
   IF ("数据块_1".二号车轮写入速度 > 1) AND ("数据块_1".二号车轮写入速度 < 33000) THEN
       "原地转向-二号车轮转换" := INT_TO_REAL("数据块_1".二号车轮写入速度);
       "原地转向-二号车轮转换" := "原地转向-二号车轮转换"*1.00474+(-10.0);
       "数据块_1"."二号车轮直行模拟量（已校准）" := ROUND("原地转向-二号车轮转换");
   END_IF;
   IF "数据块_1".二号车轮写入速度 = 0 THEN "数据块_1"."二号车轮直行模拟量（已校准）" := 0; END_IF;
END_REGION

REGION Network 3
   // 1.0015 15
   // 1.0 0
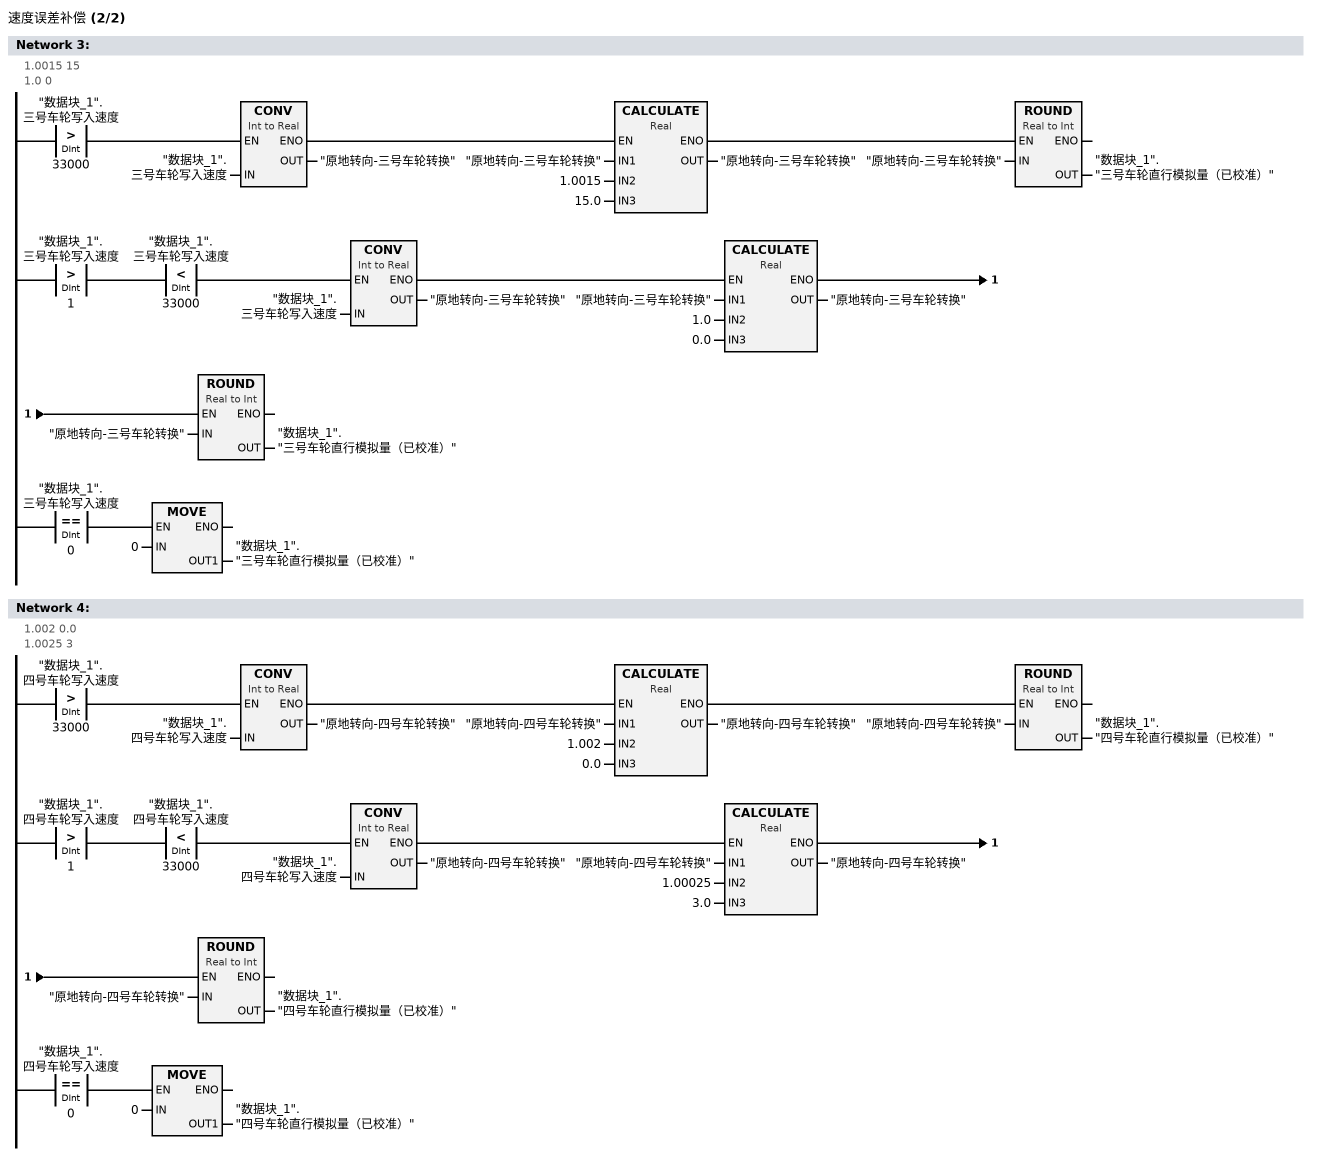
   RUNG wire#powerrail
      { S7_Templates := "SrcType := DInt" } GT_Contact(in1 := "数据块_1".三号车轮写入速度, in2 := 33000)
      { S7_Templates := "[SrcType := Int, DestType := Real]" } Convert(in := "数据块_1".三号车轮写入速度, out => "原地转向-三号车轮转换")
      { S7_Templates := "SrcType := Real"; S7_Expression := "IN1*IN2+IN3" } Calculate(in1 := "原地转向-三号车轮转换", in2 := 1.0015, in3 := 15.0, out => "原地转向-三号车轮转换")
      { S7_Templates := "[SrcType := Real, DestType := Int]" } Round(in := "原地转向-三号车轮转换", out => "数据块_1"."三号车轮直行模拟量（已校准）")
   END_RUNG
   RUNG wire#powerrail
      { S7_Templates := "SrcType := DInt" } GT_Contact(in1 := "数据块_1".三号车轮写入速度, in2 := 1)
      { S7_Templates := "SrcType := DInt" } LT_Contact(in1 := "数据块_1".三号车轮写入速度, in2 := 33000)
      { S7_Templates := "[SrcType := Int, DestType := Real]" } Convert(in := "数据块_1".三号车轮写入速度, out => "原地转向-三号车轮转换")
      { S7_Templates := "SrcType := Real"; S7_Expression := "IN1*IN2+IN3" } Calculate(in1 := "原地转向-三号车轮转换", in2 := 1.0, in3 := 0.0, out => "原地转向-三号车轮转换")
      { S7_Templates := "[SrcType := Real, DestType := Int]" } Round(in := "原地转向-三号车轮转换", out => "数据块_1"."三号车轮直行模拟量（已校准）")
   END_RUNG
   RUNG wire#powerrail
      { S7_Templates := "SrcType := DInt" } EQ_Contact(in1 := "数据块_1".三号车轮写入速度, in2 := 0)
      Move(in := 0, out1 => "数据块_1"."三号车轮直行模拟量（已校准）")
   END_RUNG
   // the same network as SCL:
   IF "数据块_1".三号车轮写入速度 > 33000 THEN
       "原地转向-三号车轮转换" := INT_TO_REAL("数据块_1".三号车轮写入速度);
       "原地转向-三号车轮转换" := "原地转向-三号车轮转换"*1.0015+15.0;
       "数据块_1"."三号车轮直行模拟量（已校准）" := ROUND("原地转向-三号车轮转换");
   END_IF;
   IF ("数据块_1".三号车轮写入速度 > 1) AND ("数据块_1".三号车轮写入速度 < 33000) THEN
       "原地转向-三号车轮转换" := INT_TO_REAL("数据块_1".三号车轮写入速度);
       "原地转向-三号车轮转换" := "原地转向-三号车轮转换"*1.0+0.0;
       "数据块_1"."三号车轮直行模拟量（已校准）" := ROUND("原地转向-三号车轮转换");
   END_IF;
   IF "数据块_1".三号车轮写入速度 = 0 THEN "数据块_1"."三号车轮直行模拟量（已校准）" := 0; END_IF;
END_REGION

REGION Network 4
   // 1.002 0.0
   // 1.0025 3
   RUNG wire#powerrail
      { S7_Templates := "SrcType := DInt" } GT_Contact(in1 := "数据块_1".四号车轮写入速度, in2 := 33000)
      { S7_Templates := "[SrcType := Int, DestType := Real]" } Convert(in := "数据块_1".四号车轮写入速度, out => "原地转向-四号车轮转换")
      { S7_Templates := "SrcType := Real"; S7_Expression := "IN1*IN2+IN3" } Calculate(in1 := "原地转向-四号车轮转换", in2 := 1.002, in3 := 0.0, out => "原地转向-四号车轮转换")
      { S7_Templates := "[SrcType := Real, DestType := Int]" } Round(in := "原地转向-四号车轮转换", out => "数据块_1"."四号车轮直行模拟量（已校准）")
   END_RUNG
   RUNG wire#powerrail
      { S7_Templates := "SrcType := DInt" } GT_Contact(in1 := "数据块_1".四号车轮写入速度, in2 := 1)
      { S7_Templates := "SrcType := DInt" } LT_Contact(in1 := "数据块_1".四号车轮写入速度, in2 := 33000)
      { S7_Templates := "[SrcType := Int, DestType := Real]" } Convert(in := "数据块_1".四号车轮写入速度, out => "原地转向-四号车轮转换")
      { S7_Templates := "SrcType := Real"; S7_Expression := "IN1*IN2+IN3" } Calculate(in1 := "原地转向-四号车轮转换", in2 := 1.00025, in3 := 3.0, out => "原地转向-四号车轮转换")
      { S7_Templates := "[SrcType := Real, DestType := Int]" } Round(in := "原地转向-四号车轮转换", out => "数据块_1"."四号车轮直行模拟量（已校准）")
   END_RUNG
   RUNG wire#powerrail
      { S7_Templates := "SrcType := DInt" } EQ_Contact(in1 := "数据块_1".四号车轮写入速度, in2 := 0)
      Move(in := 0, out1 => "数据块_1"."四号车轮直行模拟量（已校准）")
   END_RUNG
   // the same network as SCL:
   IF "数据块_1".四号车轮写入速度 > 33000 THEN
       "原地转向-四号车轮转换" := INT_TO_REAL("数据块_1".四号车轮写入速度);
       "原地转向-四号车轮转换" := "原地转向-四号车轮转换"*1.002+0.0;
       "数据块_1"."四号车轮直行模拟量（已校准）" := ROUND("原地转向-四号车轮转换");
   END_IF;
   IF ("数据块_1".四号车轮写入速度 > 1) AND ("数据块_1".四号车轮写入速度 < 33000) THEN
       "原地转向-四号车轮转换" := INT_TO_REAL("数据块_1".四号车轮写入速度);
       "原地转向-四号车轮转换" := "原地转向-四号车轮转换"*1.00025+3.0;
       "数据块_1"."四号车轮直行模拟量（已校准）" := ROUND("原地转向-四号车轮转换");
   END_IF;
   IF "数据块_1".四号车轮写入速度 = 0 THEN "数据块_1"."四号车轮直行模拟量（已校准）" := 0; END_IF;
END_REGION
END_FUNCTION

FUNCTION "回零点" : Void   // FC10, LAD
{ S7_Optimized_Access := 'TRUE' }
VERSION : 0.1
BEGIN

REGION Network 1
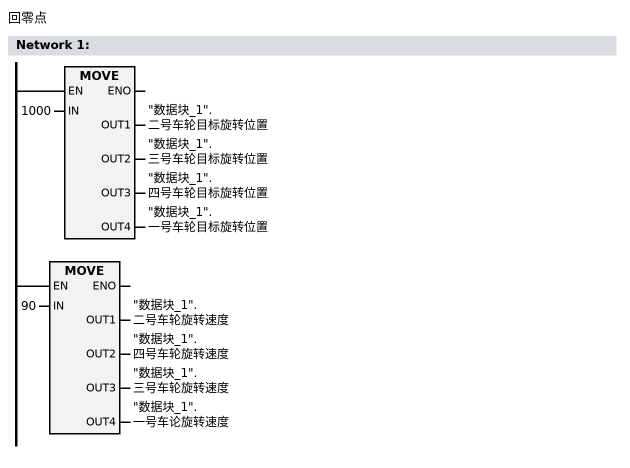
   RUNG wire#powerrail
      Move(in := 1000, out1 => "数据块_1".二号车轮目标旋转位置, out2 => "数据块_1".三号车轮目标旋转位置, out3 => "数据块_1".四号车轮目标旋转位置, out4 => "数据块_1".一号车轮目标旋转位置)
   END_RUNG
   RUNG wire#powerrail
      Move(in := 90, out1 => "数据块_1".二号车轮旋转速度, out2 => "数据块_1".四号车轮旋转速度, out3 => "数据块_1".三号车轮旋转速度, out4 => "数据块_1".一号车论旋转速度)
   END_RUNG
   // the same network as SCL:
   "数据块_1".二号车轮目标旋转位置 := 1000;
   "数据块_1".三号车轮目标旋转位置 := 1000;
   "数据块_1".四号车轮目标旋转位置 := 1000;
   "数据块_1".一号车轮目标旋转位置 := 1000;
   "数据块_1".二号车轮旋转速度 := 90;
   "数据块_1".四号车轮旋转速度 := 90;
   "数据块_1".三号车轮旋转速度 := 90;
   "数据块_1".一号车论旋转速度 := 90;
END_REGION
END_FUNCTION

ORGANIZATION_BLOCK "Main"   // OB1, LAD, ProgramCycle
TITLE = "Main Program Sweep (Cycle)"
{ S7_Optimized_Access := 'TRUE' }
VERSION : 0.1
   VAR_INPUT
      Initial_Call : Bool;   // Initial call of this OB
      Remanence : Bool;   // =True, if remanent data are available
   END_VAR
BEGIN

REGION Network 1
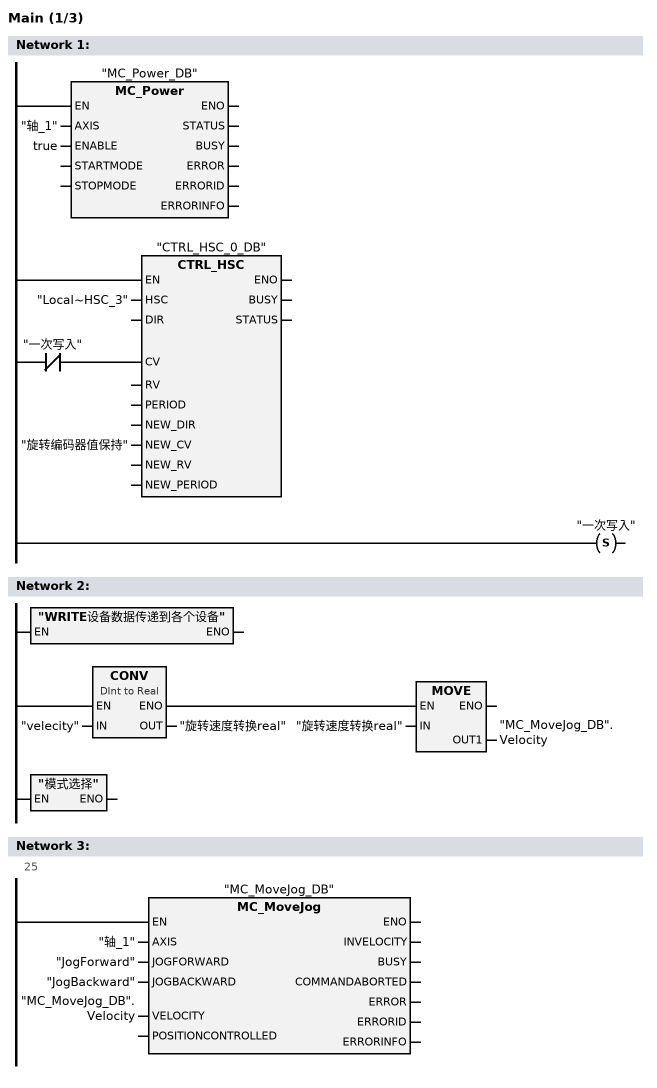
   "MC_Power_DB"(Axis := "轴_1", Enable := true);   // MC_Power
   "CTRL_HSC_0_DB"(HSC := "Local~HSC_3", CV := NOT "一次写入", NEW_CV := "旋转编码器值保持");   // CTRL_HSC
   "一次写入" := TRUE;
END_REGION

REGION Network 2
   RUNG wire#powerrail
      "WRITE设备数据传递到各个设备"()
   END_RUNG
   RUNG wire#powerrail
      { S7_Templates := "[SrcType := DInt, DestType := Real]" } Convert(in := "velecity", out => "旋转速度转换real")
      Move(in := "旋转速度转换real", out1 => "MC_MoveJog_DB".Velocity)
   END_RUNG
   RUNG wire#powerrail
      "模式选择"()
   END_RUNG
   // the same network as SCL:
   "WRITE设备数据传递到各个设备"();
   "旋转速度转换real" := DINT_TO_REAL("velecity");
   "MC_MoveJog_DB".Velocity := "旋转速度转换real";
   "模式选择"();
END_REGION

REGION Network 3
   // 25
   "MC_MoveJog_DB"(Axis := "轴_1",   // MC_MoveJog
                   JogForward := "JogForward",
                   JogBackward := "JogBackward",
                   Velocity := "MC_MoveJog_DB".Velocity);
END_REGION

REGION Network 4
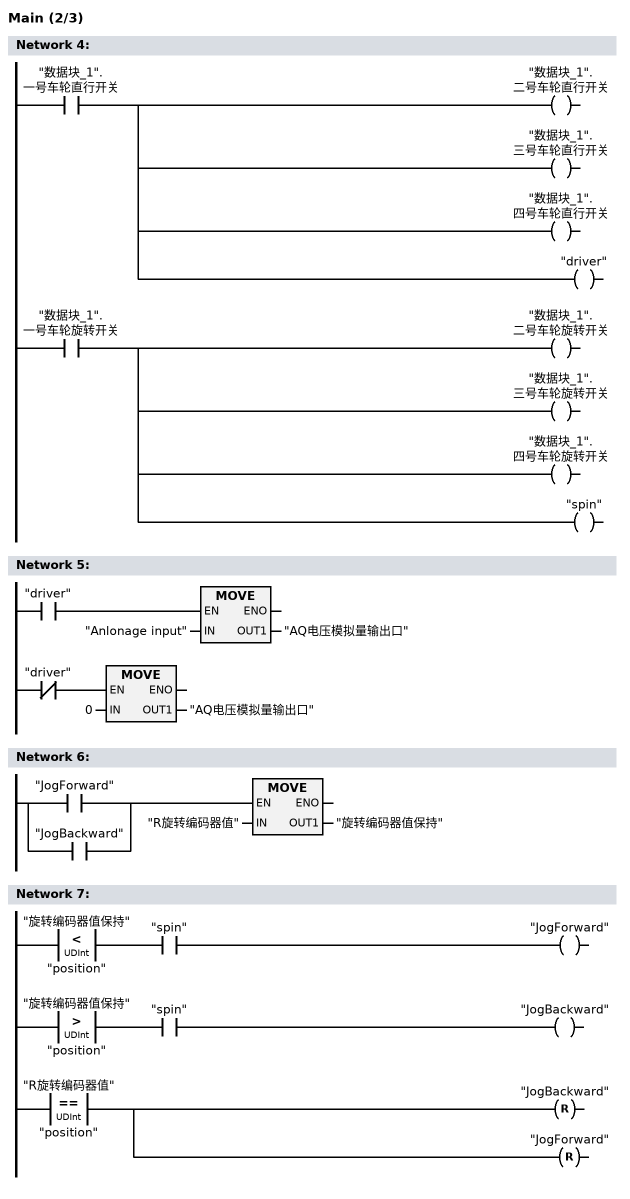
   RUNG wire#powerrail
      Contact( "数据块_1".一号车轮直行开关 )
      wire#w1
      Coil( "数据块_1".二号车轮直行开关 )
   END_RUNG
   RUNG wire#w1
      Coil( "数据块_1".三号车轮直行开关 )
   END_RUNG
   RUNG wire#w1
      Coil( "数据块_1".四号车轮直行开关 )
   END_RUNG
   RUNG wire#w1
      Coil( "driver" )
   END_RUNG
   RUNG wire#powerrail
      Contact( "数据块_1".一号车轮旋转开关 )
      wire#w2
      Coil( "数据块_1".二号车轮旋转开关 )
   END_RUNG
   RUNG wire#w2
      Coil( "数据块_1".三号车轮旋转开关 )
   END_RUNG
   RUNG wire#w2
      Coil( "数据块_1".四号车轮旋转开关 )
   END_RUNG
   RUNG wire#w2
      Coil( "spin" )
   END_RUNG
   // the same network as SCL:
   "数据块_1".二号车轮直行开关 := "数据块_1".一号车轮直行开关;
   "数据块_1".三号车轮直行开关 := "数据块_1".一号车轮直行开关;
   "数据块_1".四号车轮直行开关 := "数据块_1".一号车轮直行开关;
   "driver" := "数据块_1".一号车轮直行开关;
   "数据块_1".二号车轮旋转开关 := "数据块_1".一号车轮旋转开关;
   "数据块_1".三号车轮旋转开关 := "数据块_1".一号车轮旋转开关;
   "数据块_1".四号车轮旋转开关 := "数据块_1".一号车轮旋转开关;
   "spin" := "数据块_1".一号车轮旋转开关;
END_REGION

REGION Network 5
   RUNG wire#powerrail
      Contact( "driver" )
      Move(in := "Anlonage input", out1 => "AQ电压模拟量输出口")
   END_RUNG
   RUNG wire#powerrail
      I_Contact( "driver" )
      Move(in := 0, out1 => "AQ电压模拟量输出口")
   END_RUNG
   // the same network as SCL:
   IF "driver" THEN "AQ电压模拟量输出口" := "Anlonage input"; END_IF;
   IF NOT "driver" THEN "AQ电压模拟量输出口" := 0; END_IF;
END_REGION

REGION Network 6
   RUNG wire#powerrail
      Contact( "JogForward" )
      wire#w1
      Move(in := "R旋转编码器值", out1 => "旋转编码器值保持")
   END_RUNG
   RUNG wire#powerrail
      Contact( "JogBackward" )
   END_RUNG wire#w1
   // the same network as SCL:
   IF "JogForward" OR "JogBackward" THEN "旋转编码器值保持" := "R旋转编码器值"; END_IF;
END_REGION

REGION Network 7
   RUNG wire#powerrail
      { S7_Templates := "SrcType := UDInt" } LT_Contact(in1 := "旋转编码器值保持", in2 := "position")
      Contact( "spin" )
      Coil( "JogForward" )
   END_RUNG
   RUNG wire#powerrail
      { S7_Templates := "SrcType := UDInt" } GT_Contact(in1 := "旋转编码器值保持", in2 := "position")
      Contact( "spin" )
      Coil( "JogBackward" )
   END_RUNG
   RUNG wire#powerrail
      { S7_Templates := "SrcType := UDInt" } EQ_Contact(in1 := "R旋转编码器值", in2 := "position")
      wire#w1
      R_Coil( "JogBackward" )
   END_RUNG
   RUNG wire#w1
      R_Coil( "JogForward" )
   END_RUNG
   // the same network as SCL:
   "JogForward" := ("旋转编码器值保持" < "position") AND "spin";
   "JogBackward" := ("旋转编码器值保持" > "position") AND "spin";
   IF "R旋转编码器值" = "position" THEN
       "JogBackward" := FALSE;
       "JogForward" := FALSE;
   END_IF;
END_REGION

REGION Network 8
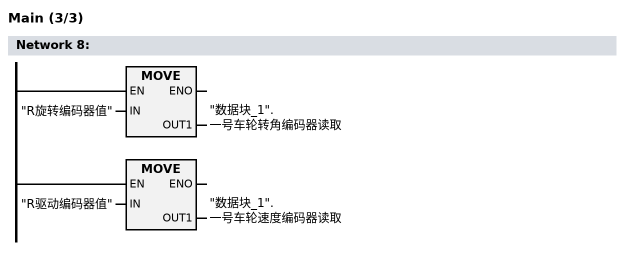
   RUNG wire#powerrail
      Move(in := "R旋转编码器值", out1 => "数据块_1".一号车轮转角编码器读取)
   END_RUNG
   RUNG wire#powerrail
      Move(in := "R驱动编码器值", out1 => "数据块_1".一号车轮速度编码器读取)
   END_RUNG
   // the same network as SCL:
   "数据块_1".一号车轮转角编码器读取 := "R旋转编码器值";
   "数据块_1".一号车轮速度编码器读取 := "R驱动编码器值";
END_REGION
END_ORGANIZATION_BLOCK

// ===== PLC "PLC_2"  CPU 1212C DC/DC/DC =====

VAR_GLOBAL   // PLC tag table "默认变量表"
   "轴_1_脉冲" AT %Q0.0 : Bool;
   "轴_1_方向" AT %Q0.1 : Bool;
   "JogForward" AT %I100.0 : Bool;
   "JogBackward" AT %I100.1 : Bool;
   "drive" AT %I200.1 : Bool;
   "AQ电压模拟量输出口" AT %QW80 : Word;
   "Anlonage input" AT %IW208 : Word;
   "旋转编码器值保持" AT %MD0 : DWord;
   "R驱动编码器值" AT %ID1000 : DWord;
   "一次写入" AT %M5.0 : Bool;
   "position" AT %IW202 : Word;
   "velecity" AT %ID204 : DWord;
   "R旋转编码器值" AT %ID1008 : DWord;
   "spin" AT %I200.0 : Bool;
   "旋转速度转换real" AT %MD24 : Real;
   "旋转传输到1号" AT %QD300 : DWord;
   "驱动传输到1号" AT %QD304 : DWord;
END_VAR

DATA_BLOCK "轴_1"   // DB2, Motion_DB
{ S7_Optimized_Access := 'TRUE' }
AUTHOR : SIMATIC
FAMILY : BasicMC
NAME : TO_PosAx
VERSION : 6.0
// stored: InstanceOfName TO_PositioningAxis
"TO_PositioningAxis"
BEGIN
   // Axis.OnlinePtoModeCU = 16#0000_0002
   // Axis.DirectionOutputEnabledCU = TRUE
   // Axis.SelectedChannel2EnumCU = %Q0.1
   // Axis.SelectedChannel1EnumCU = %Q0.0
   // Pulse.MinDeltaDeltaFrequencyCU = 0.004
   // Pulse.MaxDeltaDeltaFrequencyCU = 1.0E+10
   // Pulse.MinDeltaFrequencyCU = 0.005
   // Pulse.MaxDeltaFrequencyCU = 9.5E+9
   // Pulse.MinFrequencyCU = 1.0
   // Pulse.MaxFrequencyCU = 100000.0
   // Pulse.OutputSourceCU = 16#0000_0000
   // Axis.SelectPTO = 0
END_DATA_BLOCK

ORGANIZATION_BLOCK "Main"   // OB1, LAD, ProgramCycle
TITLE = "Main Program Sweep (Cycle)"
{ S7_Optimized_Access := 'TRUE' }
VERSION : 0.1
   VAR_INPUT
      Initial_Call : Bool;   // Initial call of this OB
      Remanence : Bool;   // =True, if remanent data are available
   END_VAR
BEGIN

REGION Network 1
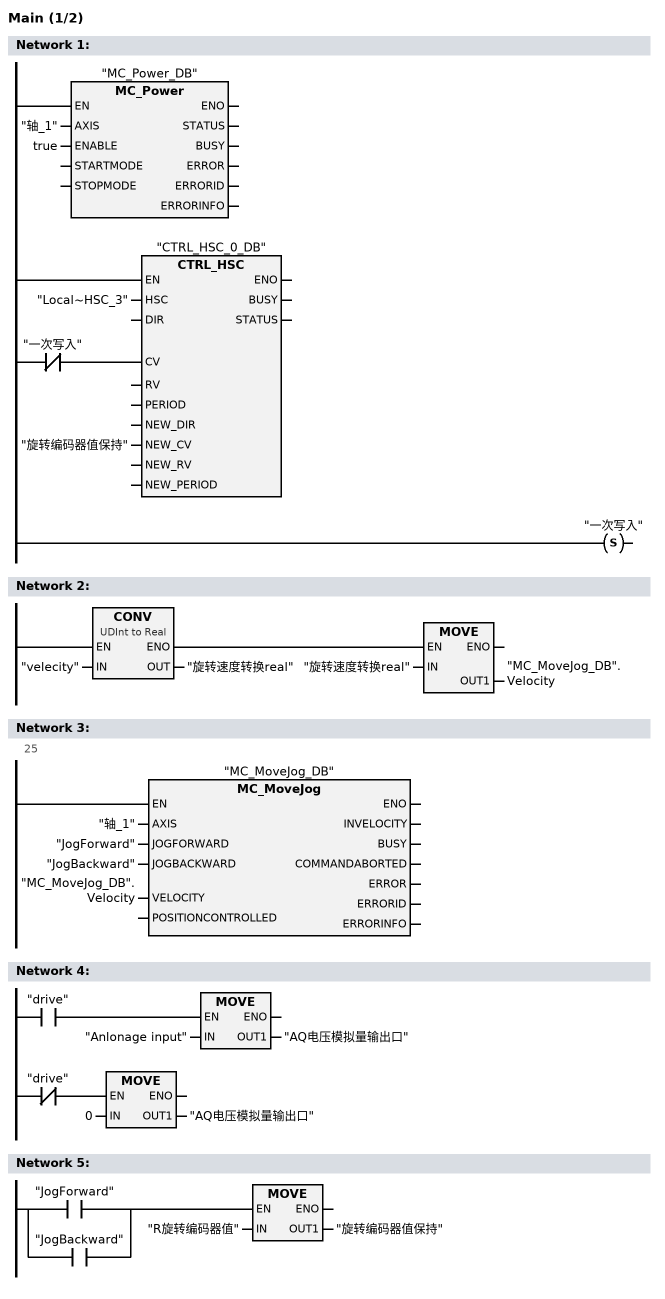
   "MC_Power_DB"(Axis := "轴_1", Enable := true);   // MC_Power
   "CTRL_HSC_0_DB"(HSC := "Local~HSC_3", CV := NOT "一次写入", NEW_CV := "旋转编码器值保持");   // CTRL_HSC
   "一次写入" := TRUE;
END_REGION

REGION Network 2
   RUNG wire#powerrail
      { S7_Templates := "[SrcType := UDInt, DestType := Real]" } Convert(in := "velecity", out => "旋转速度转换real")
      Move(in := "旋转速度转换real", out1 => "MC_MoveJog_DB".Velocity)
   END_RUNG
   // the same network as SCL:
   "旋转速度转换real" := UDINT_TO_REAL("velecity");
   "MC_MoveJog_DB".Velocity := "旋转速度转换real";
END_REGION

REGION Network 3
   // 25
   "MC_MoveJog_DB"(Axis := "轴_1",   // MC_MoveJog
                   JogForward := "JogForward",
                   JogBackward := "JogBackward",
                   Velocity := "MC_MoveJog_DB".Velocity);
END_REGION

REGION Network 4
   RUNG wire#powerrail
      Contact( "drive" )
      Move(in := "Anlonage input", out1 => "AQ电压模拟量输出口")
   END_RUNG
   RUNG wire#powerrail
      I_Contact( "drive" )
      Move(in := 0, out1 => "AQ电压模拟量输出口")
   END_RUNG
   // the same network as SCL:
   IF "drive" THEN "AQ电压模拟量输出口" := "Anlonage input"; END_IF;
   IF NOT "drive" THEN "AQ电压模拟量输出口" := 0; END_IF;
END_REGION

REGION Network 5
   RUNG wire#powerrail
      Contact( "JogForward" )
      wire#w1
      Move(in := "R旋转编码器值", out1 => "旋转编码器值保持")
   END_RUNG
   RUNG wire#powerrail
      Contact( "JogBackward" )
   END_RUNG wire#w1
   // the same network as SCL:
   IF "JogForward" OR "JogBackward" THEN "旋转编码器值保持" := "R旋转编码器值"; END_IF;
END_REGION

REGION Network 6
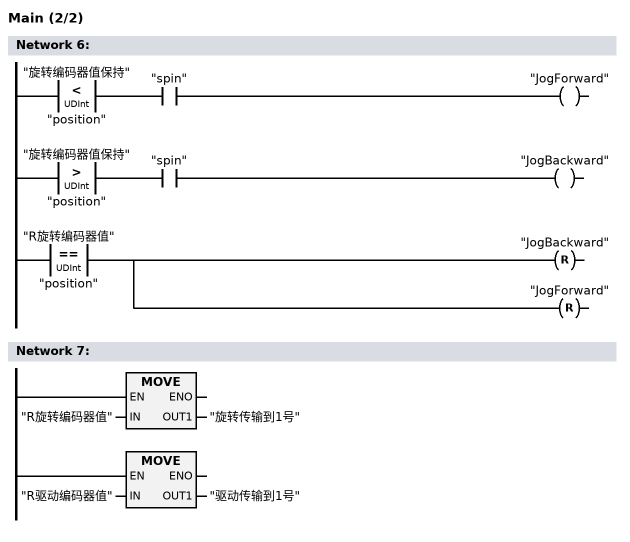
   RUNG wire#powerrail
      { S7_Templates := "SrcType := UDInt" } LT_Contact(in1 := "旋转编码器值保持", in2 := "position")
      Contact( "spin" )
      Coil( "JogForward" )
   END_RUNG
   RUNG wire#powerrail
      { S7_Templates := "SrcType := UDInt" } GT_Contact(in1 := "旋转编码器值保持", in2 := "position")
      Contact( "spin" )
      Coil( "JogBackward" )
   END_RUNG
   RUNG wire#powerrail
      { S7_Templates := "SrcType := UDInt" } EQ_Contact(in1 := "R旋转编码器值", in2 := "position")
      wire#w1
      R_Coil( "JogBackward" )
   END_RUNG
   RUNG wire#w1
      R_Coil( "JogForward" )
   END_RUNG
   // the same network as SCL:
   "JogForward" := ("旋转编码器值保持" < "position") AND "spin";
   "JogBackward" := ("旋转编码器值保持" > "position") AND "spin";
   IF "R旋转编码器值" = "position" THEN
       "JogBackward" := FALSE;
       "JogForward" := FALSE;
   END_IF;
END_REGION

REGION Network 7
   RUNG wire#powerrail
      Move(in := "R旋转编码器值", out1 => "旋转传输到1号")
   END_RUNG
   RUNG wire#powerrail
      Move(in := "R驱动编码器值", out1 => "驱动传输到1号")
   END_RUNG
   // the same network as SCL:
   "旋转传输到1号" := "R旋转编码器值";
   "驱动传输到1号" := "R驱动编码器值";
END_REGION
END_ORGANIZATION_BLOCK

// ===== PLC "PLC_3"  CPU 1212C DC/DC/DC =====

VAR_GLOBAL   // PLC tag table "默认变量表"
   "轴_1_脉冲" AT %Q0.0 : Bool;
   "轴_1_方向" AT %Q0.1 : Bool;
   "JogForward" AT %I100.0 : Bool;
   "JogBackward" AT %I100.1 : Bool;
   "drive" AT %I200.1 : Bool;
   "AQ电压模拟量输出口" AT %QW80 : Word;
   "Anlonage input" AT %IW208 : Word;
   "旋转编码器值保持" AT %MD0 : DWord;
   "R驱动编码器值" AT %ID1000 : DWord;
   "一次写入" AT %M5.0 : Bool;
   "position" AT %IW202 : Word;
   "velecity" AT %ID204 : DWord;
   "R旋转编码器值" AT %ID1008 : DWord;
   "spin" AT %I200.0 : Bool;
   "旋转速度转换real" AT %MD24 : Real;
   "旋转传输到1号" AT %QD300 : DWord;
   "驱动传输到1号" AT %QD304 : DWord;
END_VAR

DATA_BLOCK "轴_1"   // DB2, Motion_DB
{ S7_Optimized_Access := 'TRUE' }
AUTHOR : SIMATIC
FAMILY : BasicMC
NAME : TO_PosAx
VERSION : 6.0
// stored: InstanceOfName TO_PositioningAxis
"TO_PositioningAxis"
BEGIN
   // Axis.OnlinePtoModeCU = 16#0000_0002
   // Axis.DirectionOutputEnabledCU = TRUE
   // Axis.SelectedChannel2EnumCU = %Q0.1
   // Axis.SelectedChannel1EnumCU = %Q0.0
   // Pulse.MinDeltaDeltaFrequencyCU = 0.004
   // Pulse.MaxDeltaDeltaFrequencyCU = 1.0E+10
   // Pulse.MinDeltaFrequencyCU = 0.005
   // Pulse.MaxDeltaFrequencyCU = 9.5E+9
   // Pulse.MinFrequencyCU = 1.0
   // Pulse.MaxFrequencyCU = 100000.0
   // Pulse.OutputSourceCU = 16#0000_0000
   // Axis.SelectPTO = 0
END_DATA_BLOCK

ORGANIZATION_BLOCK "Main"   // OB1, LAD, ProgramCycle
TITLE = "Main Program Sweep (Cycle)"
{ S7_Optimized_Access := 'TRUE' }
VERSION : 0.1
   VAR_INPUT
      Initial_Call : Bool;   // Initial call of this OB
      Remanence : Bool;   // =True, if remanent data are available
   END_VAR
BEGIN

REGION Network 1
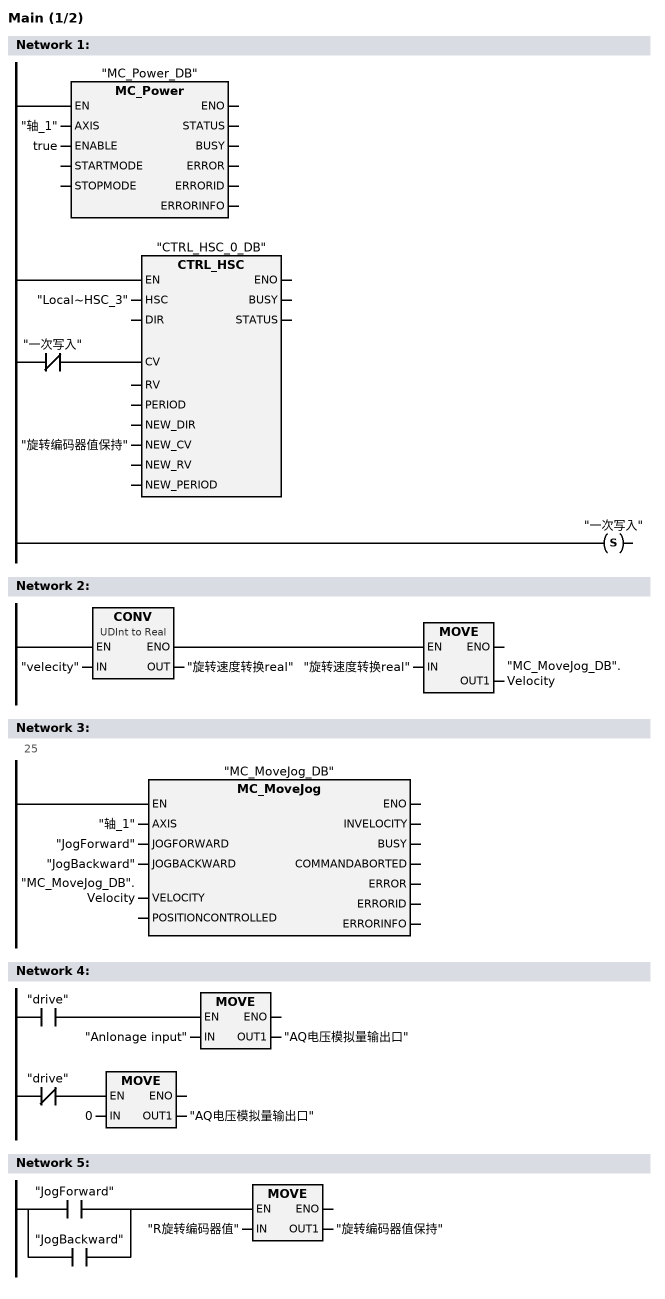
   "MC_Power_DB"(Axis := "轴_1", Enable := true);   // MC_Power
   "CTRL_HSC_0_DB"(HSC := "Local~HSC_3", CV := NOT "一次写入", NEW_CV := "旋转编码器值保持");   // CTRL_HSC
   "一次写入" := TRUE;
END_REGION

REGION Network 2
   RUNG wire#powerrail
      { S7_Templates := "[SrcType := UDInt, DestType := Real]" } Convert(in := "velecity", out => "旋转速度转换real")
      Move(in := "旋转速度转换real", out1 => "MC_MoveJog_DB".Velocity)
   END_RUNG
   // the same network as SCL:
   "旋转速度转换real" := UDINT_TO_REAL("velecity");
   "MC_MoveJog_DB".Velocity := "旋转速度转换real";
END_REGION

REGION Network 3
   // 25
   "MC_MoveJog_DB"(Axis := "轴_1",   // MC_MoveJog
                   JogForward := "JogForward",
                   JogBackward := "JogBackward",
                   Velocity := "MC_MoveJog_DB".Velocity);
END_REGION

REGION Network 4
   RUNG wire#powerrail
      Contact( "drive" )
      Move(in := "Anlonage input", out1 => "AQ电压模拟量输出口")
   END_RUNG
   RUNG wire#powerrail
      I_Contact( "drive" )
      Move(in := 0, out1 => "AQ电压模拟量输出口")
   END_RUNG
   // the same network as SCL:
   IF "drive" THEN "AQ电压模拟量输出口" := "Anlonage input"; END_IF;
   IF NOT "drive" THEN "AQ电压模拟量输出口" := 0; END_IF;
END_REGION

REGION Network 5
   RUNG wire#powerrail
      Contact( "JogForward" )
      wire#w1
      Move(in := "R旋转编码器值", out1 => "旋转编码器值保持")
   END_RUNG
   RUNG wire#powerrail
      Contact( "JogBackward" )
   END_RUNG wire#w1
   // the same network as SCL:
   IF "JogForward" OR "JogBackward" THEN "旋转编码器值保持" := "R旋转编码器值"; END_IF;
END_REGION

REGION Network 6
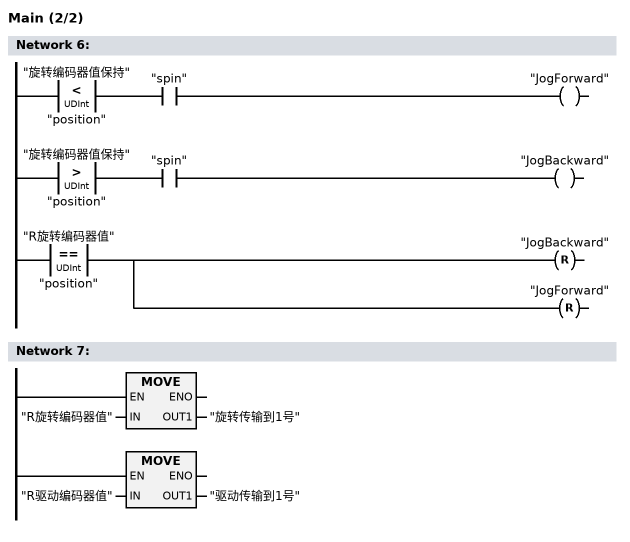
   RUNG wire#powerrail
      { S7_Templates := "SrcType := UDInt" } LT_Contact(in1 := "旋转编码器值保持", in2 := "position")
      Contact( "spin" )
      Coil( "JogForward" )
   END_RUNG
   RUNG wire#powerrail
      { S7_Templates := "SrcType := UDInt" } GT_Contact(in1 := "旋转编码器值保持", in2 := "position")
      Contact( "spin" )
      Coil( "JogBackward" )
   END_RUNG
   RUNG wire#powerrail
      { S7_Templates := "SrcType := UDInt" } EQ_Contact(in1 := "R旋转编码器值", in2 := "position")
      wire#w1
      R_Coil( "JogBackward" )
   END_RUNG
   RUNG wire#w1
      R_Coil( "JogForward" )
   END_RUNG
   // the same network as SCL:
   "JogForward" := ("旋转编码器值保持" < "position") AND "spin";
   "JogBackward" := ("旋转编码器值保持" > "position") AND "spin";
   IF "R旋转编码器值" = "position" THEN
       "JogBackward" := FALSE;
       "JogForward" := FALSE;
   END_IF;
END_REGION

REGION Network 7
   RUNG wire#powerrail
      Move(in := "R旋转编码器值", out1 => "旋转传输到1号")
   END_RUNG
   RUNG wire#powerrail
      Move(in := "R驱动编码器值", out1 => "驱动传输到1号")
   END_RUNG
   // the same network as SCL:
   "旋转传输到1号" := "R旋转编码器值";
   "驱动传输到1号" := "R驱动编码器值";
END_REGION
END_ORGANIZATION_BLOCK

// ===== PLC "PLC_4"  CPU 1212C DC/DC/DC =====

VAR_GLOBAL   // PLC tag table "默认变量表"
   "轴_1_脉冲" AT %Q0.0 : Bool;
   "轴_1_方向" AT %Q0.1 : Bool;
   "JogForward" AT %I100.0 : Bool;
   "JogBackward" AT %I100.1 : Bool;
   "drive" AT %I200.1 : Bool;
   "AQ电压模拟量输出口" AT %QW80 : Word;
   "Anlonage input" AT %IW208 : Word;
   "旋转编码器值保持" AT %MD0 : DWord;
   "R驱动编码器值" AT %ID1000 : DWord;
   "一次写入" AT %M5.0 : Bool;
   "position" AT %IW202 : Word;
   "velecity" AT %ID204 : DWord;
   "R旋转编码器值" AT %ID1008 : DWord;
   "spin" AT %I200.0 : Bool;
   "旋转速度转换real" AT %MD24 : Real;
   "旋转传输到1号" AT %QD300 : DWord;
   "驱动传输到1号" AT %QD304 : DWord;
END_VAR

DATA_BLOCK "轴_1"   // DB2, Motion_DB
{ S7_Optimized_Access := 'TRUE' }
AUTHOR : SIMATIC
FAMILY : BasicMC
NAME : TO_PosAx
VERSION : 6.0
// stored: InstanceOfName TO_PositioningAxis
"TO_PositioningAxis"
BEGIN
   // Axis.OnlinePtoModeCU = 16#0000_0002
   // Axis.DirectionOutputEnabledCU = TRUE
   // Axis.SelectedChannel2EnumCU = %Q0.1
   // Axis.SelectedChannel1EnumCU = %Q0.0
   // Pulse.MinDeltaDeltaFrequencyCU = 0.004
   // Pulse.MaxDeltaDeltaFrequencyCU = 1.0E+10
   // Pulse.MinDeltaFrequencyCU = 0.005
   // Pulse.MaxDeltaFrequencyCU = 9.5E+9
   // Pulse.MinFrequencyCU = 1.0
   // Pulse.MaxFrequencyCU = 100000.0
   // Pulse.OutputSourceCU = 16#0000_0000
   // Axis.SelectPTO = 0
END_DATA_BLOCK

ORGANIZATION_BLOCK "Main"   // OB1, LAD, ProgramCycle
TITLE = "Main Program Sweep (Cycle)"
{ S7_Optimized_Access := 'TRUE' }
VERSION : 0.1
   VAR_INPUT
      Initial_Call : Bool;   // Initial call of this OB
      Remanence : Bool;   // =True, if remanent data are available
   END_VAR
BEGIN

REGION Network 1
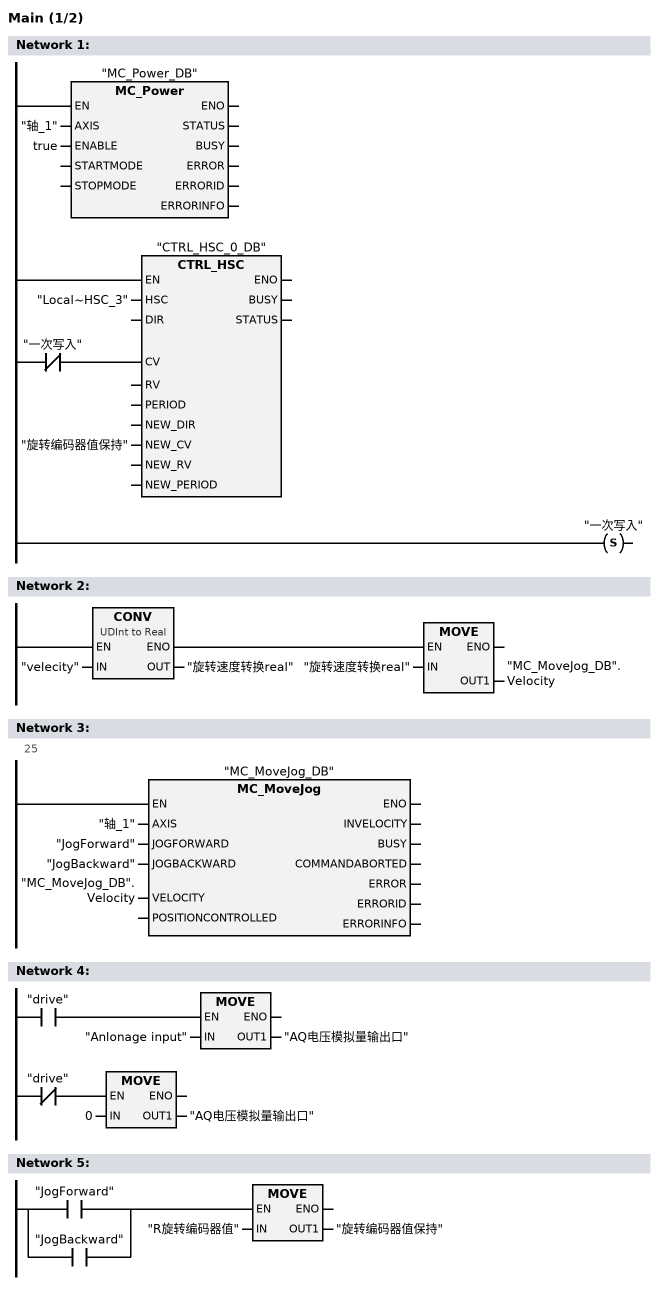
   "MC_Power_DB"(Axis := "轴_1", Enable := true);   // MC_Power
   "CTRL_HSC_0_DB"(HSC := "Local~HSC_3", CV := NOT "一次写入", NEW_CV := "旋转编码器值保持");   // CTRL_HSC
   "一次写入" := TRUE;
END_REGION

REGION Network 2
   RUNG wire#powerrail
      { S7_Templates := "[SrcType := UDInt, DestType := Real]" } Convert(in := "velecity", out => "旋转速度转换real")
      Move(in := "旋转速度转换real", out1 => "MC_MoveJog_DB".Velocity)
   END_RUNG
   // the same network as SCL:
   "旋转速度转换real" := UDINT_TO_REAL("velecity");
   "MC_MoveJog_DB".Velocity := "旋转速度转换real";
END_REGION

REGION Network 3
   // 25
   "MC_MoveJog_DB"(Axis := "轴_1",   // MC_MoveJog
                   JogForward := "JogForward",
                   JogBackward := "JogBackward",
                   Velocity := "MC_MoveJog_DB".Velocity);
END_REGION

REGION Network 4
   RUNG wire#powerrail
      Contact( "drive" )
      Move(in := "Anlonage input", out1 => "AQ电压模拟量输出口")
   END_RUNG
   RUNG wire#powerrail
      I_Contact( "drive" )
      Move(in := 0, out1 => "AQ电压模拟量输出口")
   END_RUNG
   // the same network as SCL:
   IF "drive" THEN "AQ电压模拟量输出口" := "Anlonage input"; END_IF;
   IF NOT "drive" THEN "AQ电压模拟量输出口" := 0; END_IF;
END_REGION

REGION Network 5
   RUNG wire#powerrail
      Contact( "JogForward" )
      wire#w1
      Move(in := "R旋转编码器值", out1 => "旋转编码器值保持")
   END_RUNG
   RUNG wire#powerrail
      Contact( "JogBackward" )
   END_RUNG wire#w1
   // the same network as SCL:
   IF "JogForward" OR "JogBackward" THEN "旋转编码器值保持" := "R旋转编码器值"; END_IF;
END_REGION

REGION Network 6
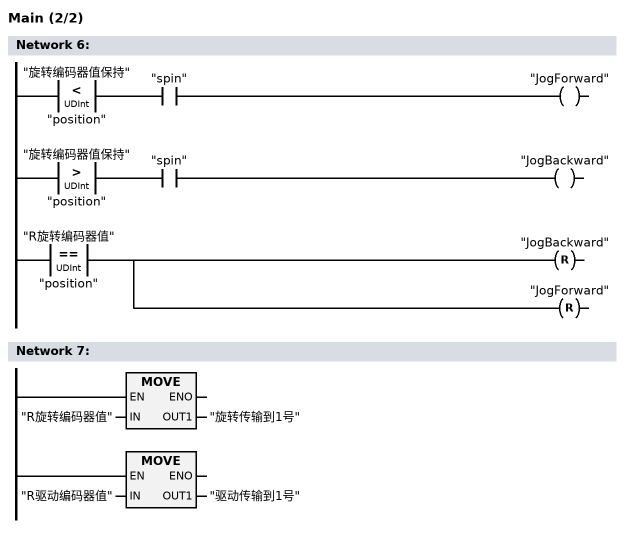
   RUNG wire#powerrail
      { S7_Templates := "SrcType := UDInt" } LT_Contact(in1 := "旋转编码器值保持", in2 := "position")
      Contact( "spin" )
      Coil( "JogForward" )
   END_RUNG
   RUNG wire#powerrail
      { S7_Templates := "SrcType := UDInt" } GT_Contact(in1 := "旋转编码器值保持", in2 := "position")
      Contact( "spin" )
      Coil( "JogBackward" )
   END_RUNG
   RUNG wire#powerrail
      { S7_Templates := "SrcType := UDInt" } EQ_Contact(in1 := "R旋转编码器值", in2 := "position")
      wire#w1
      R_Coil( "JogBackward" )
   END_RUNG
   RUNG wire#w1
      R_Coil( "JogForward" )
   END_RUNG
   // the same network as SCL:
   "JogForward" := ("旋转编码器值保持" < "position") AND "spin";
   "JogBackward" := ("旋转编码器值保持" > "position") AND "spin";
   IF "R旋转编码器值" = "position" THEN
       "JogBackward" := FALSE;
       "JogForward" := FALSE;
   END_IF;
END_REGION

REGION Network 7
   RUNG wire#powerrail
      Move(in := "R旋转编码器值", out1 => "旋转传输到1号")
   END_RUNG
   RUNG wire#powerrail
      Move(in := "R驱动编码器值", out1 => "驱动传输到1号")
   END_RUNG
   // the same network as SCL:
   "旋转传输到1号" := "R旋转编码器值";
   "驱动传输到1号" := "R驱动编码器值";
END_REGION
END_ORGANIZATION_BLOCK